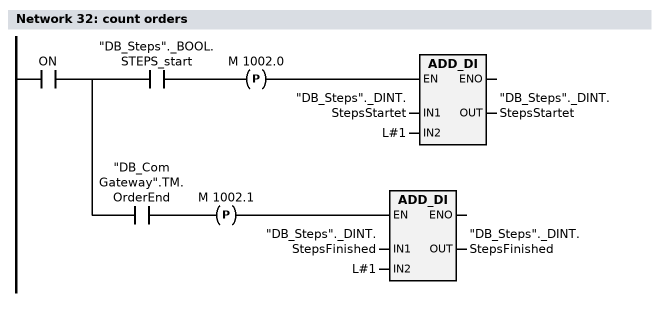
[picture p261: STEPS_OrderData networks 32-32]
NETWORK
TITLE = count orders
      A     "ON";
      =     L 35.0;
      A     L 35.0;
      A(;
      A     "DB_Steps"._BOOL.STEPS_start;
      BLD   100;
      FP    M 1002.0;
      );
      JNB   _01d;
      L     "DB_Steps"._DINT.StepsStartet;
      L     L#1;
      +D;
      T     "DB_Steps"._DINT.StepsStartet;
_01d: NOP   0;
      A     L 35.0;
      A(;
      A     "DB_ComGateway".TM.OrderEnd;
      BLD   100;
      FP    M 1002.1;
      );
      JNB   _01e;
      L     "DB_Steps"._DINT.StepsFinished;
      L     L#1;
      +D;
      T     "DB_Steps"._DINT.StepsFinished;
_01e: NOP   0;
END_FUNCTION

FUNCTION "STEPS_BASEPOS" : VOID	// FC 112
TITLE = Steps BasePos
VERSION : 0.1
BEGIN
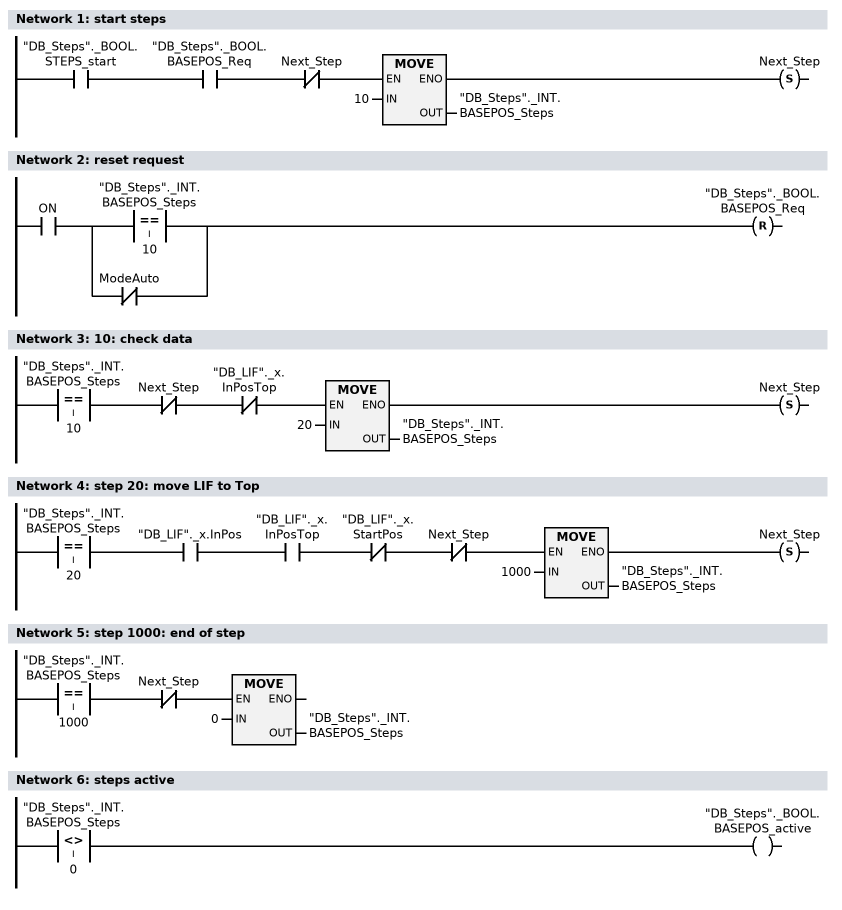
NETWORK
TITLE = start steps
      A     "DB_Steps"._BOOL.STEPS_start;
      A     "DB_Steps"._BOOL.BASEPOS_Req;
      AN    "Next_Step";
      JNB   _001;
      L     10;
      T     "DB_Steps"._INT.BASEPOS_Steps;
      SET;
      SAVE;
      CLR;
_001: A     BR;
      S     "Next_Step";
NETWORK
TITLE = reset request
      A     "ON";
      A(;
      O(;
      L     "DB_Steps"._INT.BASEPOS_Steps;
      L     10;
      ==I;
      );
      ON    "ModeAuto";
      );
      R     "DB_Steps"._BOOL.BASEPOS_Req;
NETWORK
TITLE = 10: check data
//20: move LIF to Top
      A(;
      L     "DB_Steps"._INT.BASEPOS_Steps;
      L     10;
      ==I;
      );
      AN    "Next_Step";
      AN    "DB_LIF"._x.InPosTop;
      JNB   _002;
      L     20;
      T     "DB_Steps"._INT.BASEPOS_Steps;
      SET;
      SAVE;
      CLR;
_002: A     BR;
      S     "Next_Step";
NETWORK
TITLE = step 20: move LIF to Top
//1000: end of steps
      A(;
      L     "DB_Steps"._INT.BASEPOS_Steps;
      L     20;
      ==I;
      );
      A     "DB_LIF"._x.InPos;
      A     "DB_LIF"._x.InPosTop;
      AN    "DB_LIF"._x.StartPos;
      AN    "Next_Step";
      JNB   _003;
      L     1000;
      T     "DB_Steps"._INT.BASEPOS_Steps;
      SET;
      SAVE;
      CLR;
_003: A     BR;
      S     "Next_Step";
NETWORK
TITLE = step 1000: end of step
      A(;
      L     "DB_Steps"._INT.BASEPOS_Steps;
      L     1000;
      ==I;
      );
      AN    "Next_Step";
      JNB   _004;
      L     0;
      T     "DB_Steps"._INT.BASEPOS_Steps;
_004: NOP   0;
NETWORK
TITLE = steps active
      L     "DB_Steps"._INT.BASEPOS_Steps;
      L     0;
      <>I;
      =     "DB_Steps"._BOOL.BASEPOS_active;
END_FUNCTION

FUNCTION "STEPS_EMPTY" : VOID	// FC 113
TITLE = Steps Empty
VERSION : 0.1
BEGIN
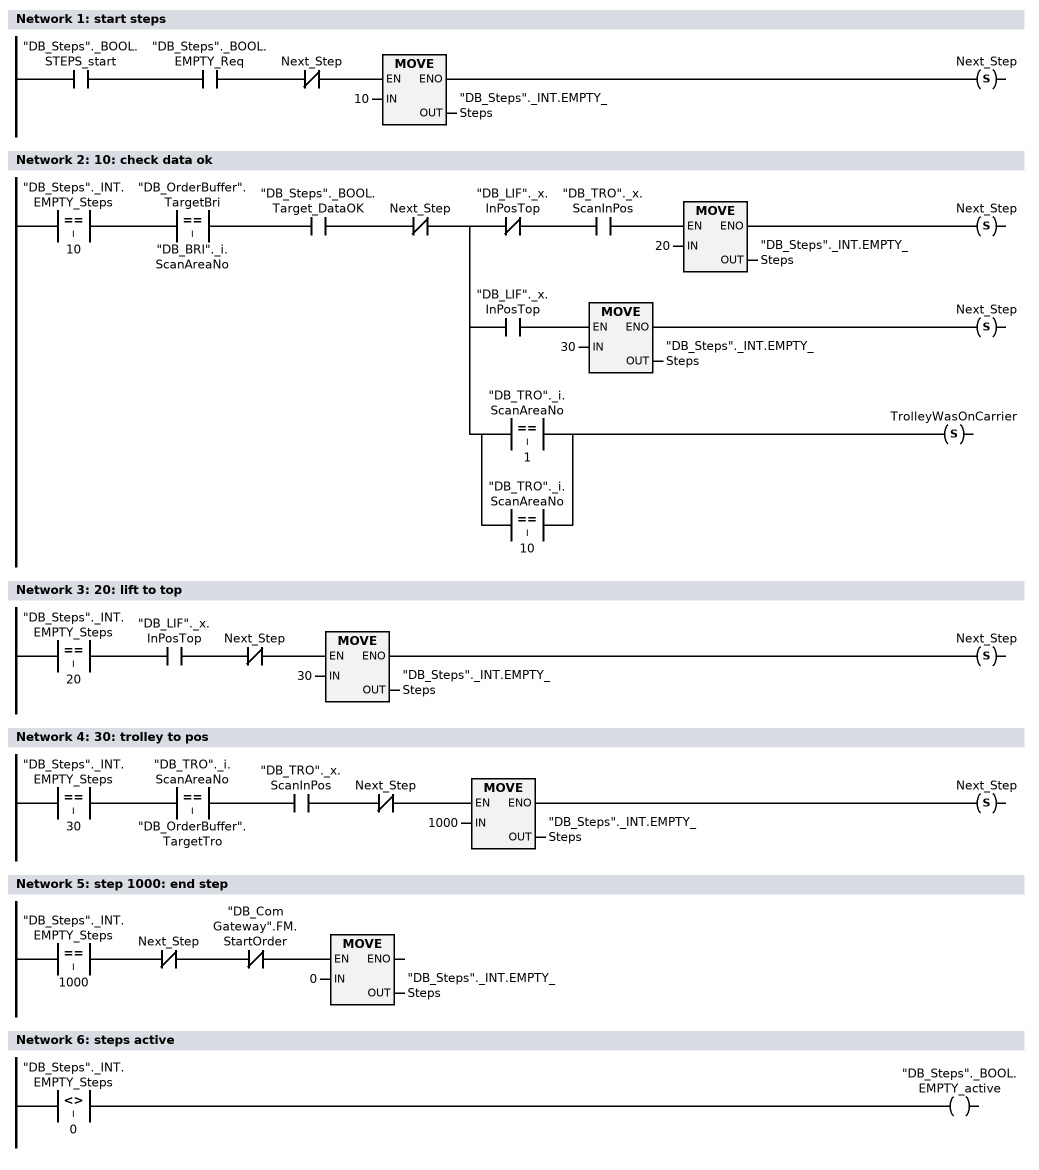
NETWORK
TITLE = start steps
      A     "DB_Steps"._BOOL.STEPS_start;
      A     "DB_Steps"._BOOL.EMPTY_Req;
      AN    "Next_Step";
      JNB   _001;
      L     10;
      T     "DB_Steps"._INT.EMPTY_Steps;
      SET;
      SAVE;
      CLR;
_001: A     BR;
      S     "Next_Step";
NETWORK
TITLE = 10: check data ok
//20: lift to top
//30: BRI to position
      A(;
      L     "DB_Steps"._INT.EMPTY_Steps;
      L     10;
      ==I;
      );
      A(;
      L     "DB_OrderBuffer".TargetBri;
      L     "DB_BRI"._i.ScanAreaNo;
      ==I;
      );
      A     "DB_Steps"._BOOL.Target_DataOK;
      AN    "Next_Step";
      =     L 0.0;
      A     L 0.0;
      AN    "DB_LIF"._x.InPosTop;
      A     "DB_TRO"._x.ScanInPos;
      JNB   _002;
      L     20;
      T     "DB_Steps"._INT.EMPTY_Steps;
      SET;
      SAVE;
      CLR;
_002: A     BR;
      S     "Next_Step";
      A     L 0.0;
      A     "DB_LIF"._x.InPosTop;
      JNB   _003;
      L     30;
      T     "DB_Steps"._INT.EMPTY_Steps;
      SET;
      SAVE;
      CLR;
_003: A     BR;
      S     "Next_Step";
      A     L 0.0;
      A(;
      O(;
      L     "DB_TRO"._i.ScanAreaNo;
      L     1;
      ==I;
      );
      O(;
      L     "DB_TRO"._i.ScanAreaNo;
      L     10;
      ==I;
      );
      );
      S     "TrolleyWasOnCarrier";
NETWORK
TITLE = 20: lift to top
//30: TRO to position
      A(;
      L     "DB_Steps"._INT.EMPTY_Steps;
      L     20;
      ==I;
      );
      A     "DB_LIF"._x.InPosTop;
      AN    "Next_Step";
      JNB   _004;
      L     30;
      T     "DB_Steps"._INT.EMPTY_Steps;
      SET;
      SAVE;
      CLR;
_004: A     BR;
      S     "Next_Step";
NETWORK
TITLE = 30: trolley to pos
      A(;
      L     "DB_Steps"._INT.EMPTY_Steps;
      L     30;
      ==I;
      );
      A(;
      L     "DB_TRO"._i.ScanAreaNo;
      L     "DB_OrderBuffer".TargetTro;
      ==I;
      );
      A     "DB_TRO"._x.ScanInPos;
      AN    "Next_Step";
      JNB   _005;
      L     1000;
      T     "DB_Steps"._INT.EMPTY_Steps;
      SET;
      SAVE;
      CLR;
_005: A     BR;
      S     "Next_Step";
NETWORK
TITLE = step 1000: end step
      A(;
      L     "DB_Steps"._INT.EMPTY_Steps;
      L     1000;
      ==I;
      );
      AN    "Next_Step";
      AN    "DB_ComGateway".FM.StartOrder;
      JNB   _006;
      L     0;
      T     "DB_Steps"._INT.EMPTY_Steps;
_006: NOP   0;
NETWORK
TITLE = steps active
      L     "DB_Steps"._INT.EMPTY_Steps;
      L     0;
      <>I;
      =     "DB_Steps"._BOOL.EMPTY_active;
END_FUNCTION

FUNCTION "STEPS_GET" : VOID	// FC 114
TITLE = Steps GET
VERSION : 0.1
VAR_TEMP
  US_Sensor_OK : BOOL ;
  GetFromLS : BOOL ;
  temp : INT ;
END_VAR
BEGIN
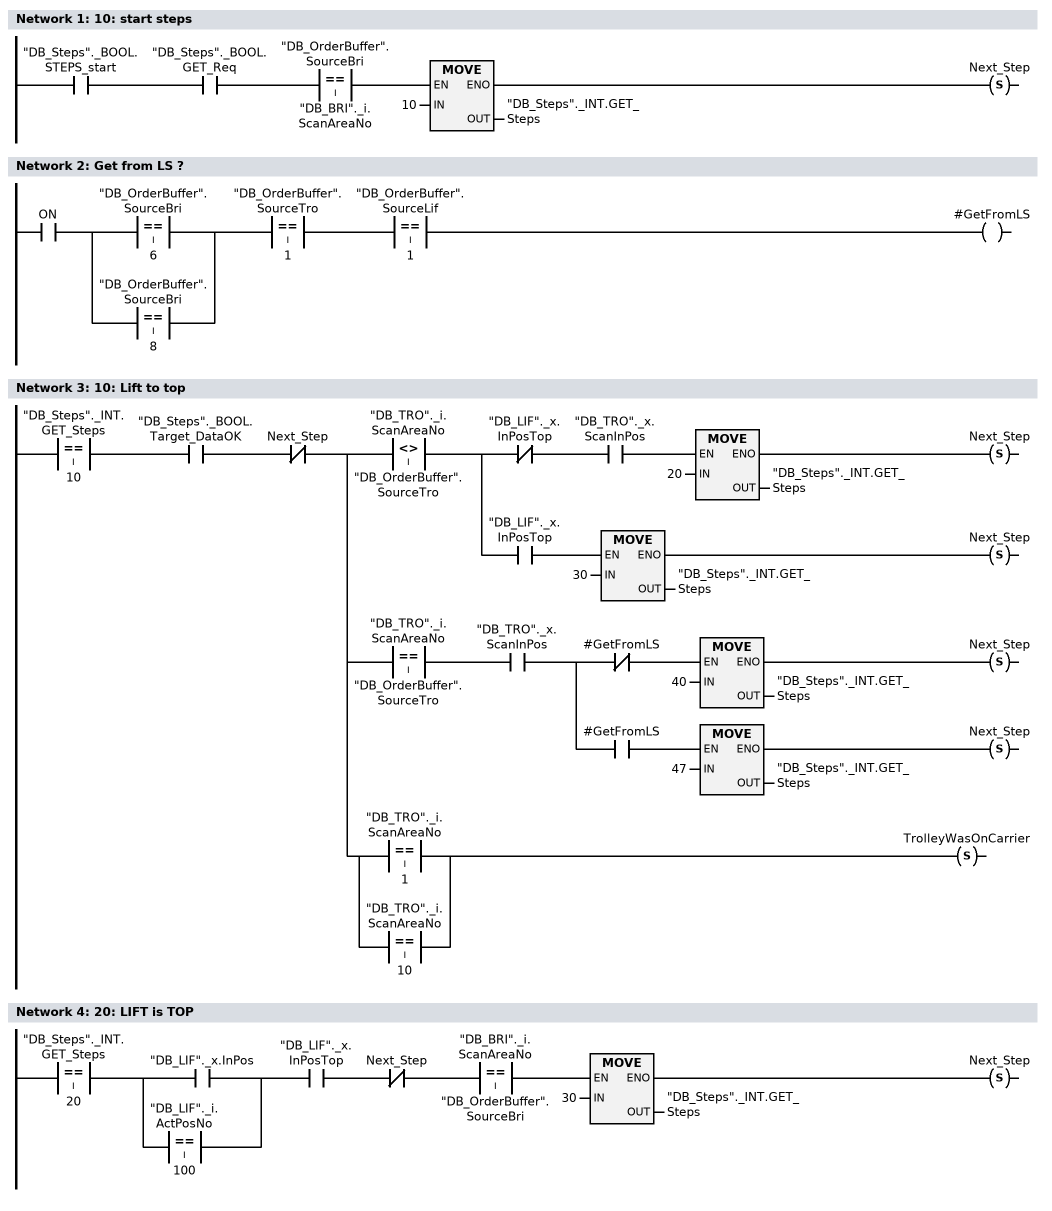
NETWORK
TITLE = 10: start steps
      A     "DB_Steps"._BOOL.STEPS_start;
      A     "DB_Steps"._BOOL.GET_Req;
      A(;
      L     "DB_OrderBuffer".SourceBri;
      L     "DB_BRI"._i.ScanAreaNo;
      ==I;
      );
      JNB   _001;
      L     10;
      T     "DB_Steps"._INT.GET_Steps;
      SET;
      SAVE;
      CLR;
_001: A     BR;
      S     "Next_Step";
NETWORK
TITLE = Get from LS ?
      A     "ON";
      A(;
      O(;
      L     "DB_OrderBuffer".SourceBri;
      L     6;
      ==I;
      );
      O(;
      L     "DB_OrderBuffer".SourceBri;
      L     8;
      ==I;
      );
      );
      A(;
      L     "DB_OrderBuffer".SourceTro;
      L     1;
      ==I;
      );
      A(;
      L     "DB_OrderBuffer".SourceLif;
      L     1;
      ==I;
      );
      =     #GetFromLS;
NETWORK
TITLE = 10: Lift to top
//20: LIF to TOP
//30: BRI to Position
      A(;
      L     "DB_Steps"._INT.GET_Steps;
      L     10;
      ==I;
      );
      A     "DB_Steps"._BOOL.Target_DataOK;
      AN    "Next_Step";
      =     L 4.0;
      A     L 4.0;
      A(;
      L     "DB_TRO"._i.ScanAreaNo;
      L     "DB_OrderBuffer".SourceTro;
      <>I;
      );
      =     L 4.1;
      A     L 4.1;
      AN    "DB_LIF"._x.InPosTop;
      A     "DB_TRO"._x.ScanInPos;
      JNB   _002;
      L     20;
      T     "DB_Steps"._INT.GET_Steps;
      SET;
      SAVE;
      CLR;
_002: A     BR;
      S     "Next_Step";
      A     L 4.1;
      A     "DB_LIF"._x.InPosTop;
      JNB   _003;
      L     30;
      T     "DB_Steps"._INT.GET_Steps;
      SET;
      SAVE;
      CLR;
_003: A     BR;
      S     "Next_Step";
      A     L 4.0;
      A(;
      L     "DB_TRO"._i.ScanAreaNo;
      L     "DB_OrderBuffer".SourceTro;
      ==I;
      );
      A     "DB_TRO"._x.ScanInPos;
      =     L 4.1;
      A     L 4.1;
      AN    #GetFromLS;
      JNB   _004;
      L     40;
      T     "DB_Steps"._INT.GET_Steps;
      SET;
      SAVE;
      CLR;
_004: A     BR;
      S     "Next_Step";
      A     L 4.1;
      A     #GetFromLS;
      JNB   _005;
      L     47;
      T     "DB_Steps"._INT.GET_Steps;
      SET;
      SAVE;
      CLR;
_005: A     BR;
      S     "Next_Step";
      A     L 4.0;
      A(;
      O(;
      L     "DB_TRO"._i.ScanAreaNo;
      L     1;
      ==I;
      );
      O(;
      L     "DB_TRO"._i.ScanAreaNo;
      L     10;
      ==I;
      );
      );
      S     "TrolleyWasOnCarrier";
NETWORK
TITLE = 20: LIFT is TOP
//30: BRI to Position / Start Width S30/S40
      A(;
      L     "DB_Steps"._INT.GET_Steps;
      L     20;
      ==I;
      );
      A(;
      O     "DB_LIF"._x.InPos;
      O(;
      L     "DB_LIF"._i.ActPosNo;
      L     100;
      ==I;
      );
      );
      A     "DB_LIF"._x.InPosTop;
      AN    "Next_Step";
      A(;
      L     "DB_BRI"._i.ScanAreaNo;
      L     "DB_OrderBuffer".SourceBri;
      ==I;
      );
      JNB   _006;
      L     30;
      T     "DB_Steps"._INT.GET_Steps;
      SET;
      SAVE;
      CLR;
_006: A     BR;
      S     "Next_Step";
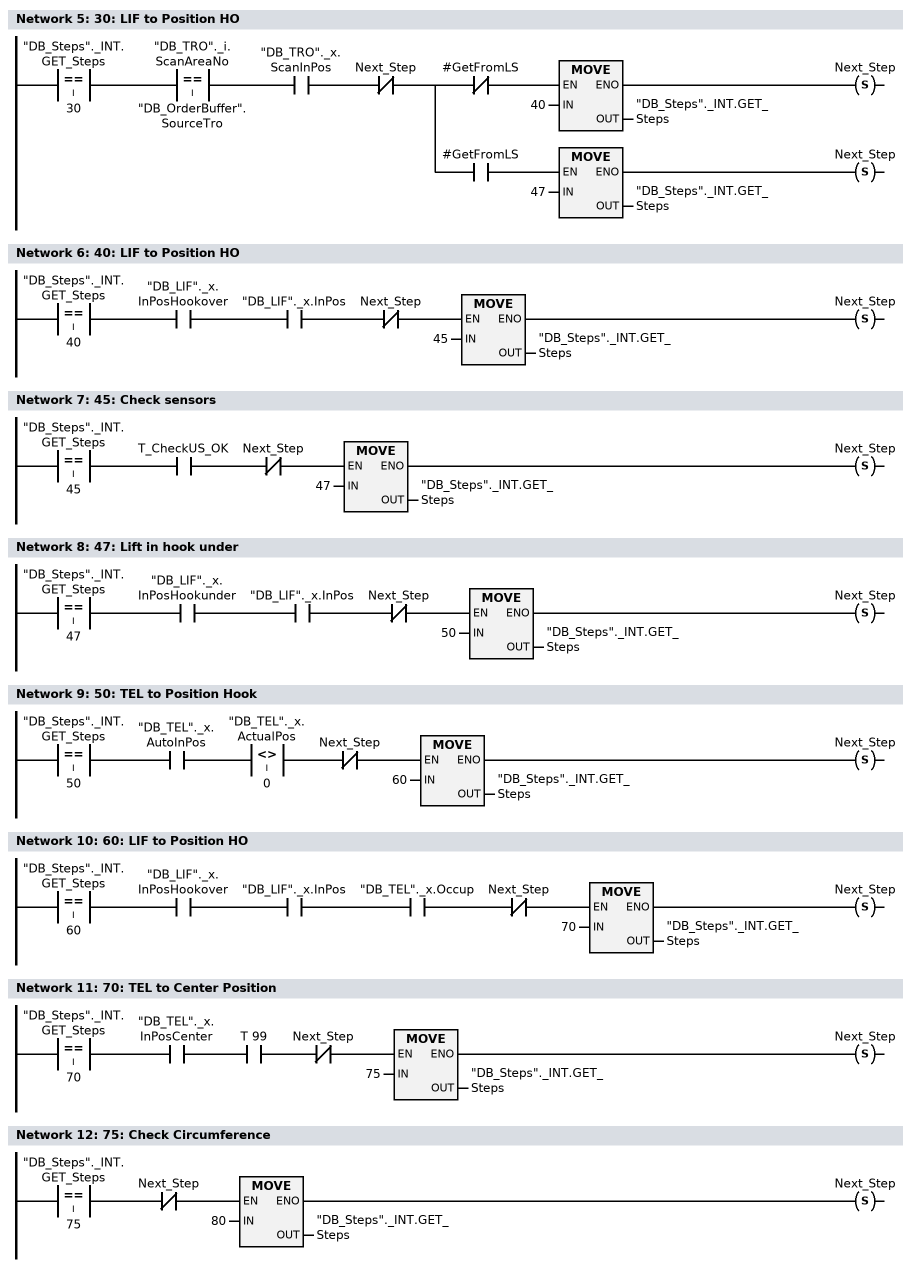
NETWORK
TITLE = 30: LIF to Position HO
      A(;
      L     "DB_Steps"._INT.GET_Steps;
      L     30;
      ==I;
      );
      A(;
      L     "DB_TRO"._i.ScanAreaNo;
      L     "DB_OrderBuffer".SourceTro;
      ==I;
      );
      A     "DB_TRO"._x.ScanInPos;
      AN    "Next_Step";
      =     L 4.0;
      A     L 4.0;
      AN    #GetFromLS;
      JNB   _007;
      L     40;
      T     "DB_Steps"._INT.GET_Steps;
      SET;
      SAVE;
      CLR;
_007: A     BR;
      S     "Next_Step";
      A     L 4.0;
      A     #GetFromLS;
      JNB   _008;
      L     47;
      T     "DB_Steps"._INT.GET_Steps;
      SET;
      SAVE;
      CLR;
_008: A     BR;
      S     "Next_Step";
NETWORK
TITLE = 40: LIF to Position HO
//50: TEL to Position Hook
//45: check occupation sensors hook over
      A(;
      L     "DB_Steps"._INT.GET_Steps;
      L     40;
      ==I;
      );
      A     "DB_LIF"._x.InPosHookover;
      A     "DB_LIF"._x.InPos;
      AN    "Next_Step";
      JNB   _009;
      L     45;
      T     "DB_Steps"._INT.GET_Steps;
      SET;
      SAVE;
      CLR;
_009: A     BR;
      S     "Next_Step";
NETWORK
TITLE = 45: Check sensors
//47: LIF to Position HU
//
//Typ 101 Lager
//Typ 201 Ladestation
//Zyp 299 Buffer
//
//The sensors are not checked on the loading staion
      A(;
      L     "DB_Steps"._INT.GET_Steps;
      L     45;
      ==I;
      );
      A     "T_CheckUS_OK";
      AN    "Next_Step";
      JNB   _00a;
      L     47;
      T     "DB_Steps"._INT.GET_Steps;
      SET;
      SAVE;
      CLR;
_00a: A     BR;
      S     "Next_Step";
NETWORK
TITLE = 47: Lift in hook under
//50: TEL to Position Hook
      A(;
      L     "DB_Steps"._INT.GET_Steps;
      L     47;
      ==I;
      );
      A     "DB_LIF"._x.InPosHookunder;
      A     "DB_LIF"._x.InPos;
      AN    "Next_Step";
      JNB   _00b;
      L     50;
      T     "DB_Steps"._INT.GET_Steps;
      SET;
      SAVE;
      CLR;
_00b: A     BR;
      S     "Next_Step";
NETWORK
TITLE = 50: TEL to Position Hook
//60: LIF to Position HO
      A(;
      L     "DB_Steps"._INT.GET_Steps;
      L     50;
      ==I;
      );
      A     "DB_TEL"._x.AutoInPos;
      A(;
      L     "DB_TEL"._x.ActualPos;
      L     0;
      <>I;
      );
      AN    "Next_Step";
      JNB   _00c;
      L     60;
      T     "DB_Steps"._INT.GET_Steps;
      SET;
      SAVE;
      CLR;
_00c: A     BR;
      S     "Next_Step";
NETWORK
TITLE = 60: LIF to Position HO
//70: TEL to Center Position
      A(;
      L     "DB_Steps"._INT.GET_Steps;
      L     60;
      ==I;
      );
      A     "DB_LIF"._x.InPosHookover;
      A     "DB_LIF"._x.InPos;
      A     "DB_TEL"._x.Occup;
      AN    "Next_Step";
      JNB   _00d;
      L     70;
      T     "DB_Steps"._INT.GET_Steps;
      SET;
      SAVE;
      CLR;
_00d: A     BR;
      S     "Next_Step";
NETWORK
TITLE = 70: TEL to Center Position
//75: Check Circumference
      A(;
      L     "DB_Steps"._INT.GET_Steps;
      L     70;
      ==I;
      );
      A     "DB_TEL"._x.InPosCenter;
      A     T 99;
      AN    "Next_Step";
      JNB   _00e;
      L     75;
      T     "DB_Steps"._INT.GET_Steps;
      SET;
      SAVE;
      CLR;
_00e: A     BR;
      S     "Next_Step";
NETWORK
TITLE = 75: Check Circumference
//510: check hook occupation sensors
// 80: check Lift position safety area loadingstation
      A(;
      L     "DB_Steps"._INT.GET_Steps;
      L     75;
      ==I;
      );
      AN    "Next_Step";
      JNB   _00f;
      L     80;
      T     "DB_Steps"._INT.GET_Steps;
      SET;
      SAVE;
      CLR;
_00f: A     BR;
      S     "Next_Step";
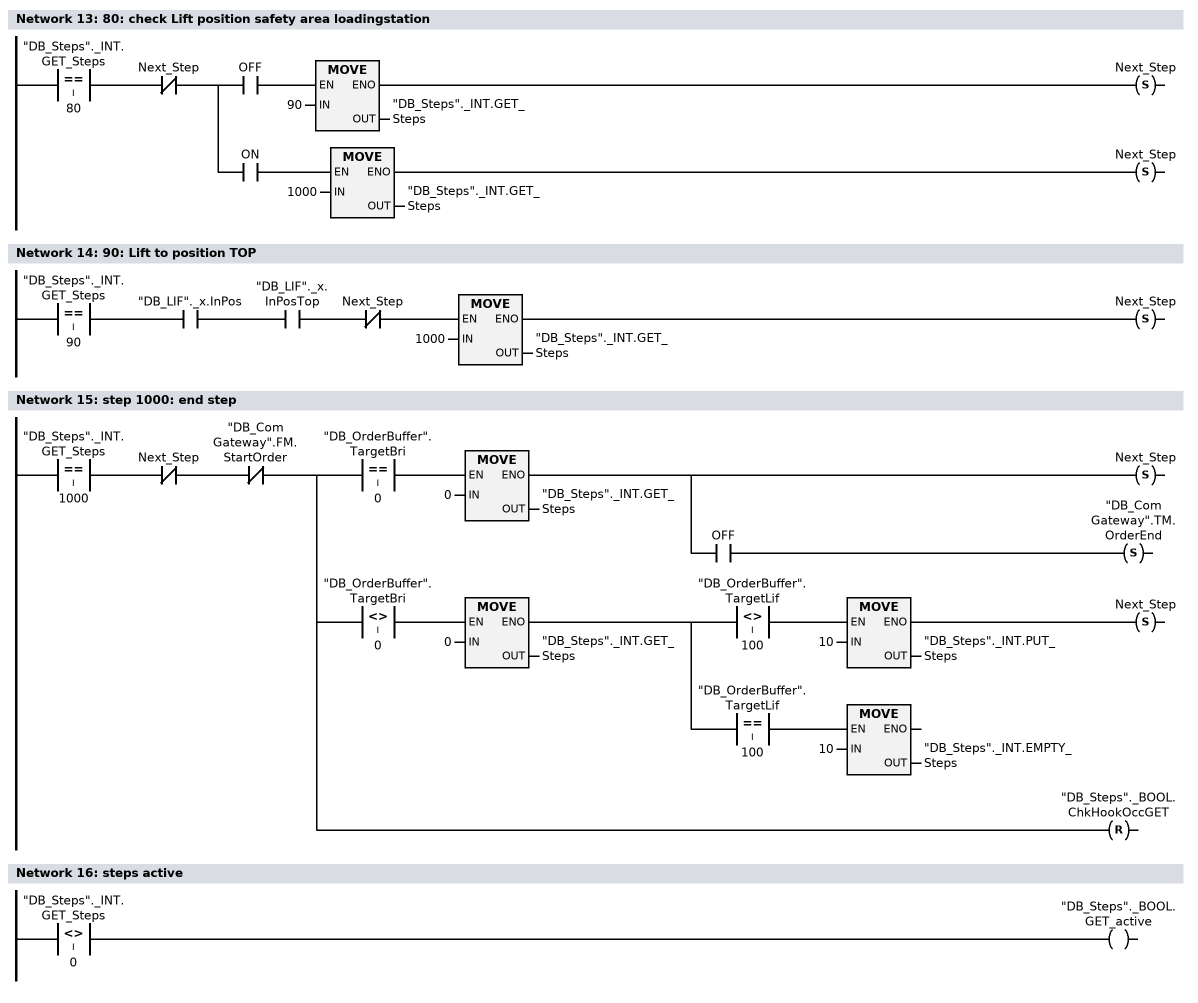
NETWORK
TITLE = 80: check Lift position safety area loadingstation
//85: Get Circumference Value
      A(;
      L     "DB_Steps"._INT.GET_Steps;
      L     80;
      ==I;
      );
      AN    "Next_Step";
      =     L 4.0;
      A     L 4.0;
      A     "OFF";
      JNB   _010;
      L     90;
      T     "DB_Steps"._INT.GET_Steps;
      SET;
      SAVE;
      CLR;
_010: A     BR;
      S     "Next_Step";
      A     L 4.0;
      A     "ON";
      JNB   _011;
      L     1000;
      T     "DB_Steps"._INT.GET_Steps;
      SET;
      SAVE;
      CLR;
_011: A     BR;
      S     "Next_Step";
NETWORK
TITLE = 90: Lift to position TOP
      A(;
      L     "DB_Steps"._INT.GET_Steps;
      L     90;
      ==I;
      );
      A     "DB_LIF"._x.InPos;
      A     "DB_LIF"._x.InPosTop;
      AN    "Next_Step";
      JNB   _012;
      L     1000;
      T     "DB_Steps"._INT.GET_Steps;
      SET;
      SAVE;
      CLR;
_012: A     BR;
      S     "Next_Step";
NETWORK
TITLE = step 1000: end step
      A(;
      L     "DB_Steps"._INT.GET_Steps;
      L     1000;
      ==I;
      );
      AN    "Next_Step";
      AN    "DB_ComGateway".FM.StartOrder;
      =     L 4.0;
      A     L 4.0;
      A(;
      L     "DB_OrderBuffer".TargetBri;
      L     0;
      ==I;
      );
      JNB   _013;
      L     0;
      T     "DB_Steps"._INT.GET_Steps;
      SET;
      SAVE;
      CLR;
_013: A     BR;
      =     L 4.1;
      A     L 4.1;
      BLD   102;
      S     "Next_Step";
      A     L 4.1;
      A     "OFF";
      S     "DB_ComGateway".TM.OrderEnd;
      A     L 4.0;
      A(;
      L     "DB_OrderBuffer".TargetBri;
      L     0;
      <>I;
      );
      JNB   _014;
      L     0;
      T     "DB_Steps"._INT.GET_Steps;
      SET;
      SAVE;
      CLR;
_014: A     BR;
      =     L 4.1;
      A     L 4.1;
      A(;
      L     "DB_OrderBuffer".TargetLif;
      L     100;
      <>I;
      );
      JNB   _015;
      L     10;
      T     "DB_Steps"._INT.PUT_Steps;
      SET;
      SAVE;
      CLR;
_015: A     BR;
      S     "Next_Step";
      A     L 4.1;
      A(;
      L     "DB_OrderBuffer".TargetLif;
      L     100;
      ==I;
      );
      JNB   _016;
      L     10;
      T     "DB_Steps"._INT.EMPTY_Steps;
_016: NOP   0;
      A     L 4.0;
      BLD   102;
      R     "DB_Steps"._BOOL.ChkHookOccGET;
NETWORK
TITLE = steps active
      L     "DB_Steps"._INT.GET_Steps;
      L     0;
      <>I;
      =     "DB_Steps"._BOOL.GET_active;
END_FUNCTION

FUNCTION "STEPS_PUT" : VOID	// FC 115
TITLE = Steps PUT
VERSION : 0.1
VAR_TEMP
  US_Sensor_OK : BOOL ;
  PutToLS : BOOL ;
  temp : INT ;
END_VAR
BEGIN
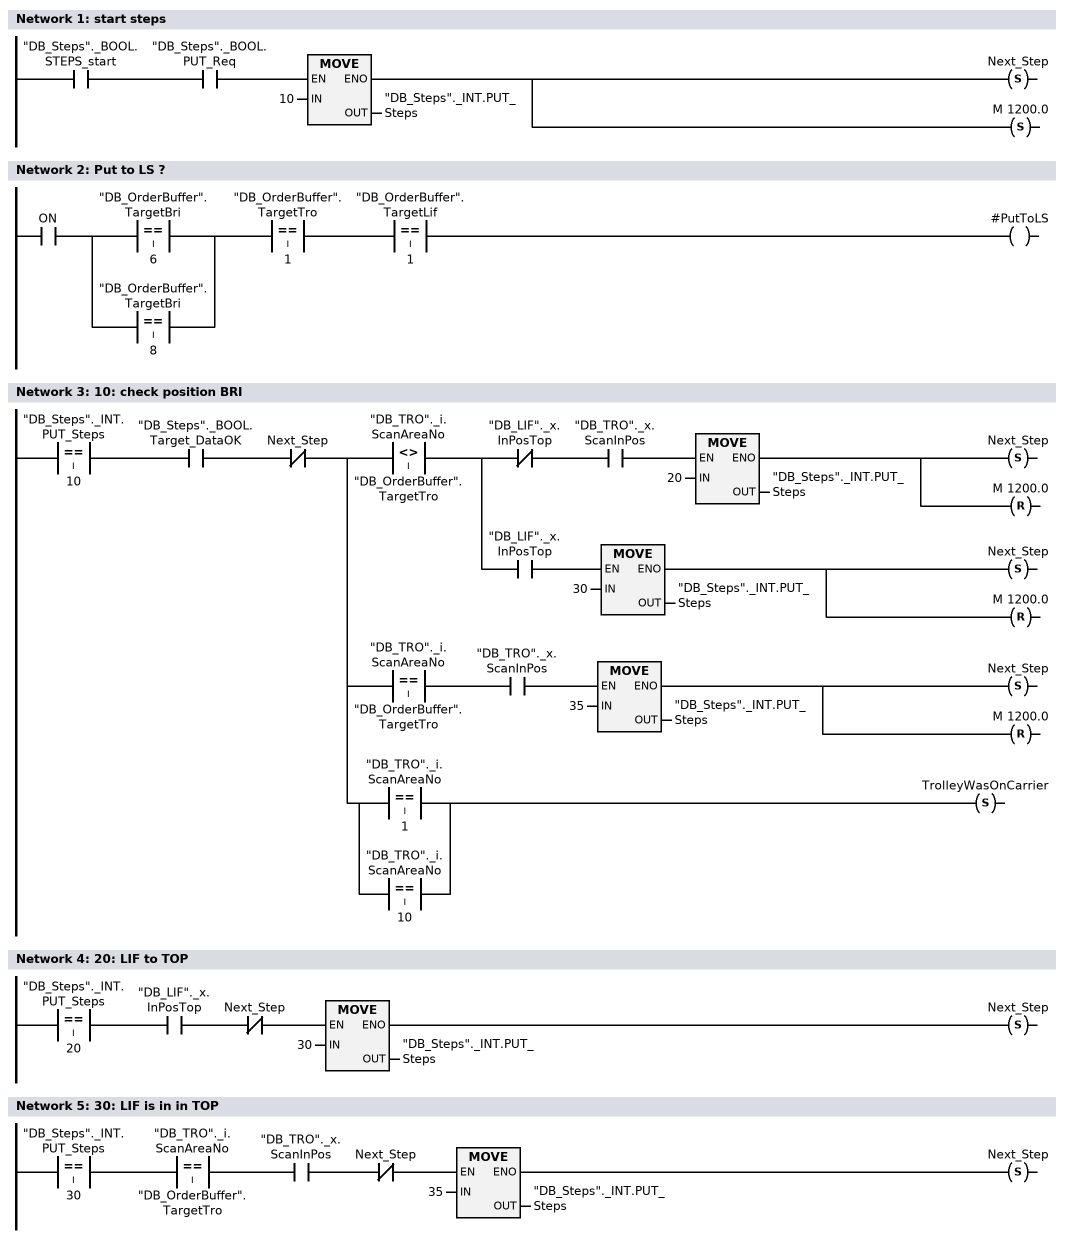
NETWORK
TITLE = start steps
      A     "DB_Steps"._BOOL.STEPS_start;
      A     "DB_Steps"._BOOL.PUT_Req;
      JNB   _001;
      L     10;
      T     "DB_Steps"._INT.PUT_Steps;
      SET;
      SAVE;
      CLR;
_001: A     BR;
      S     "Next_Step";
      S     M 1200.0;
NETWORK
TITLE = Put to LS ?
      A     "ON";
      A(;
      O(;
      L     "DB_OrderBuffer".TargetBri;
      L     6;
      ==I;
      );
      O(;
      L     "DB_OrderBuffer".TargetBri;
      L     8;
      ==I;
      );
      );
      A(;
      L     "DB_OrderBuffer".TargetTro;
      L     1;
      ==I;
      );
      A(;
      L     "DB_OrderBuffer".TargetLif;
      L     1;
      ==I;
      );
      =     #PutToLS;
NETWORK
TITLE = 10: check position BRI
//20: LIF to TOP
//30: BRI to Position
      A(;
      L     "DB_Steps"._INT.PUT_Steps;
      L     10;
      ==I;
      );
      A     "DB_Steps"._BOOL.Target_DataOK;
      AN    "Next_Step";
      =     L 4.0;
      A     L 4.0;
      A(;
      L     "DB_TRO"._i.ScanAreaNo;
      L     "DB_OrderBuffer".TargetTro;
      <>I;
      );
      =     L 4.1;
      A     L 4.1;
      AN    "DB_LIF"._x.InPosTop;
      A     "DB_TRO"._x.ScanInPos;
      JNB   _002;
      L     20;
      T     "DB_Steps"._INT.PUT_Steps;
      SET;
      SAVE;
      CLR;
_002: A     BR;
      S     "Next_Step";
      R     M 1200.0;
      A     L 4.1;
      A     "DB_LIF"._x.InPosTop;
      JNB   _003;
      L     30;
      T     "DB_Steps"._INT.PUT_Steps;
      SET;
      SAVE;
      CLR;
_003: A     BR;
      S     "Next_Step";
      R     M 1200.0;
      A     L 4.0;
      A(;
      L     "DB_TRO"._i.ScanAreaNo;
      L     "DB_OrderBuffer".TargetTro;
      ==I;
      );
      A     "DB_TRO"._x.ScanInPos;
      JNB   _004;
      L     35;
      T     "DB_Steps"._INT.PUT_Steps;
      SET;
      SAVE;
      CLR;
_004: A     BR;
      S     "Next_Step";
      R     M 1200.0;
      A     L 4.0;
      A(;
      O(;
      L     "DB_TRO"._i.ScanAreaNo;
      L     1;
      ==I;
      );
      O(;
      L     "DB_TRO"._i.ScanAreaNo;
      L     10;
      ==I;
      );
      );
      S     "TrolleyWasOnCarrier";
NETWORK
TITLE = 20: LIF to TOP
//30: BRI to Position
      A(;
      L     "DB_Steps"._INT.PUT_Steps;
      L     20;
      ==I;
      );
      A     "DB_LIF"._x.InPosTop;
      AN    "Next_Step";
      JNB   _005;
      L     30;
      T     "DB_Steps"._INT.PUT_Steps;
      SET;
      SAVE;
      CLR;
_005: A     BR;
      S     "Next_Step";
NETWORK
TITLE = 30: LIF is in in TOP
//35: LIF to Position HO
      A(;
      L     "DB_Steps"._INT.PUT_Steps;
      L     30;
      ==I;
      );
      A(;
      L     "DB_TRO"._i.ScanAreaNo;
      L     "DB_OrderBuffer".TargetTro;
      ==I;
      );
      A     "DB_TRO"._x.ScanInPos;
      AN    "Next_Step";
      JNB   _006;
      L     35;
      T     "DB_Steps"._INT.PUT_Steps;
      SET;
      SAVE;
      CLR;
_006: A     BR;
      S     "Next_Step";
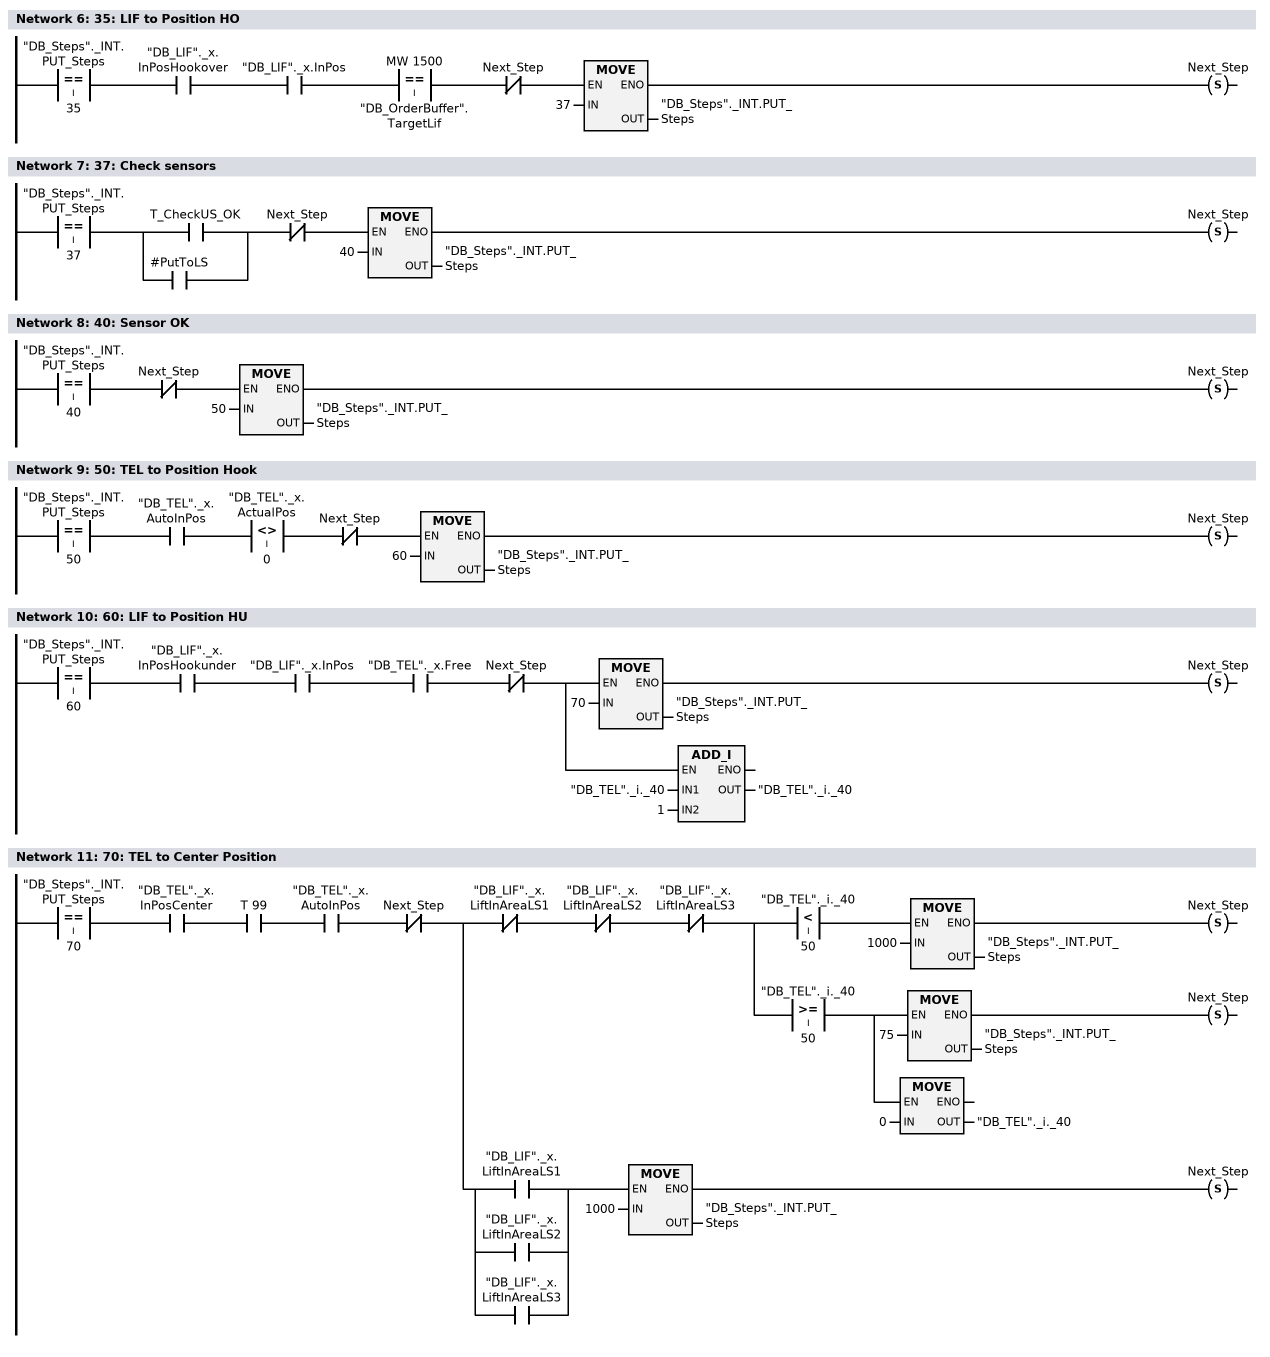
NETWORK
TITLE = 35: LIF to Position HO
//50: TEL to Position Hook
      A(;
      L     "DB_Steps"._INT.PUT_Steps;
      L     35;
      ==I;
      );
      A     "DB_LIF"._x.InPosHookover;
      A     "DB_LIF"._x.InPos;
      A(;
      L     MW 1500;
      L     "DB_OrderBuffer".TargetLif;
      ==I;
      );
      AN    "Next_Step";
      JNB   _007;
      L     37;
      T     "DB_Steps"._INT.PUT_Steps;
      SET;
      SAVE;
      CLR;
_007: A     BR;
      S     "Next_Step";
NETWORK
TITLE = 37: Check sensors
//50: TEL to Position Hook
      A(;
      L     "DB_Steps"._INT.PUT_Steps;
      L     37;
      ==I;
      );
      A(;
      O     "T_CheckUS_OK";
      O     #PutToLS;
      );
      AN    "Next_Step";
      JNB   _008;
      L     40;
      T     "DB_Steps"._INT.PUT_Steps;
      SET;
      SAVE;
      CLR;
_008: A     BR;
      S     "Next_Step";
NETWORK
TITLE = 40: Sensor OK
//50: TEL to Position Hook
      A(;
      L     "DB_Steps"._INT.PUT_Steps;
      L     40;
      ==I;
      );
      AN    "Next_Step";
      JNB   _009;
      L     50;
      T     "DB_Steps"._INT.PUT_Steps;
      SET;
      SAVE;
      CLR;
_009: A     BR;
      S     "Next_Step";
NETWORK
TITLE = 50: TEL to Position Hook
//60: LIF to Position HU
      A(;
      L     "DB_Steps"._INT.PUT_Steps;
      L     50;
      ==I;
      );
      A     "DB_TEL"._x.AutoInPos;
      A(;
      L     "DB_TEL"._x.ActualPos;
      L     0;
      <>I;
      );
      AN    "Next_Step";
      JNB   _00a;
      L     60;
      T     "DB_Steps"._INT.PUT_Steps;
      SET;
      SAVE;
      CLR;
_00a: A     BR;
      S     "Next_Step";
NETWORK
TITLE = 60: LIF to Position HU
//70: TEL to Center Position
      A(;
      L     "DB_Steps"._INT.PUT_Steps;
      L     60;
      ==I;
      );
      A     "DB_LIF"._x.InPosHookunder;
      A     "DB_LIF"._x.InPos;
      A     "DB_TEL"._x.Free;
      AN    "Next_Step";
      =     L 4.0;
      A     L 4.0;
      JNB   _00b;
      L     70;
      T     "DB_Steps"._INT.PUT_Steps;
      SET;
      SAVE;
      CLR;
_00b: A     BR;
      S     "Next_Step";
      A     L 4.0;
      JNB   _00c;
      L     "DB_TEL"._i._40;
      L     1;
      +I;
      T     "DB_TEL"._i._40;
_00c: NOP   0;
NETWORK
TITLE = 70: TEL to Center Position
//75: check occupation sensors hook
      A(;
      L     "DB_Steps"._INT.PUT_Steps;
      L     70;
      ==I;
      );
      A     "DB_TEL"._x.InPosCenter;
      A     T 99;
      A     "DB_TEL"._x.AutoInPos;
      AN    "Next_Step";
      =     L 4.0;
      A     L 4.0;
      AN    "DB_LIF"._x.LiftInAreaLS1;
      AN    "DB_LIF"._x.LiftInAreaLS2;
      AN    "DB_LIF"._x.LiftInAreaLS3;
      =     L 4.1;
      A     L 4.1;
      A(;
      L     "DB_TEL"._i._40;
      L     50;
      <I;
      );
      JNB   _00d;
      L     1000;
      T     "DB_Steps"._INT.PUT_Steps;
      SET;
      SAVE;
      CLR;
_00d: A     BR;
      S     "Next_Step";
      A     L 4.1;
      A(;
      L     "DB_TEL"._i._40;
      L     50;
      >=I;
      );
      =     L 4.2;
      A     L 4.2;
      JNB   _00e;
      L     75;
      T     "DB_Steps"._INT.PUT_Steps;
      SET;
      SAVE;
      CLR;
_00e: A     BR;
      S     "Next_Step";
      A     L 4.2;
      JNB   _00f;
      L     0;
      T     "DB_TEL"._i._40;
_00f: NOP   0;
      A     L 4.0;
      A(;
      O     "DB_LIF"._x.LiftInAreaLS1;
      O     "DB_LIF"._x.LiftInAreaLS2;
      O     "DB_LIF"._x.LiftInAreaLS3;
      );
      JNB   _010;
      L     1000;
      T     "DB_Steps"._INT.PUT_Steps;
      SET;
      SAVE;
      CLR;
_010: A     BR;
      S     "Next_Step";
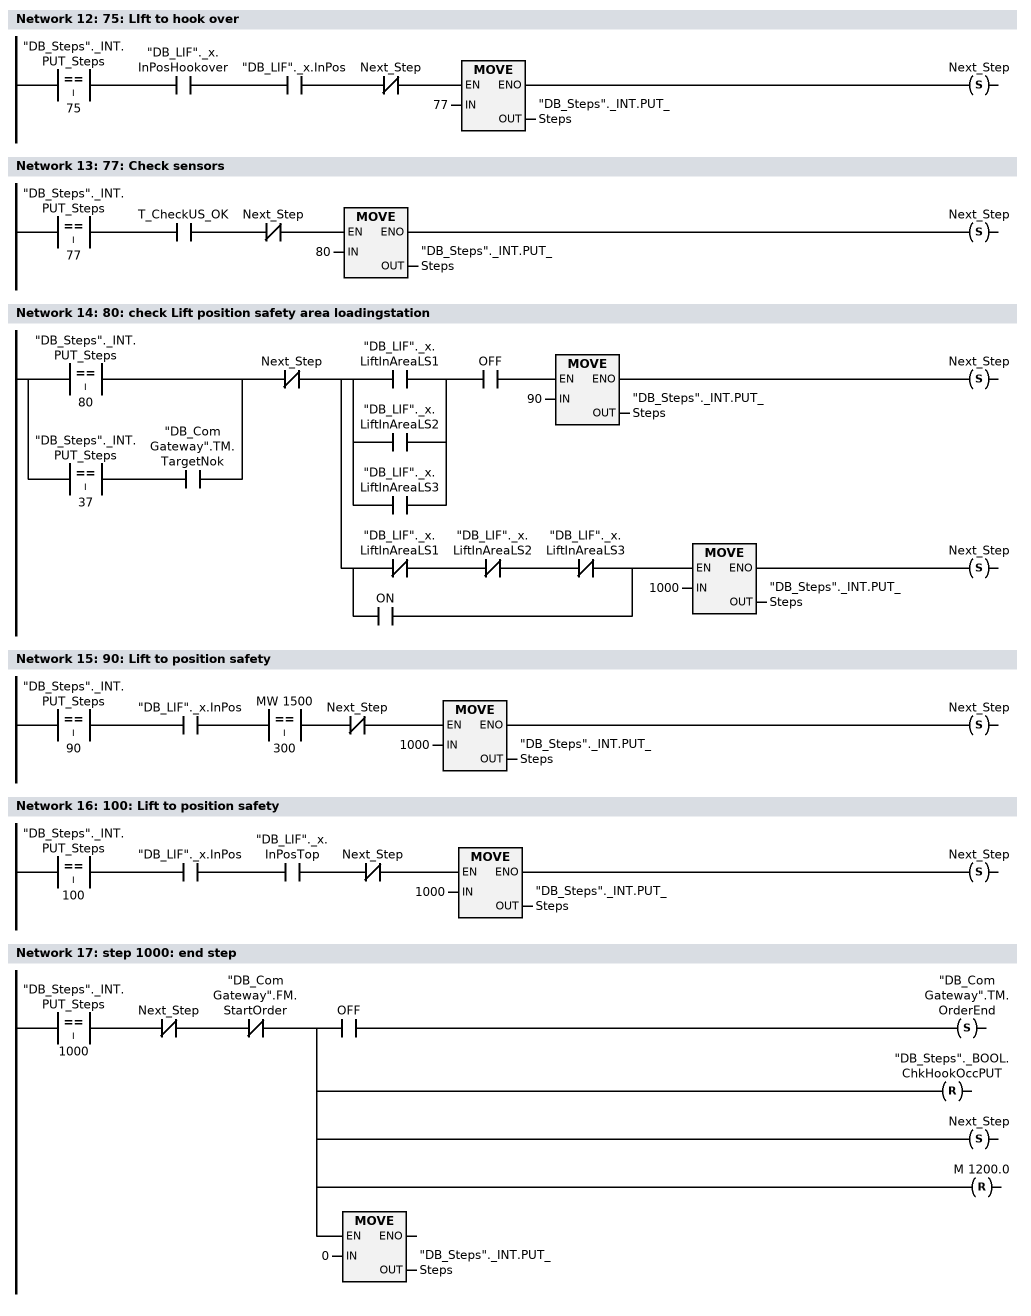
NETWORK
TITLE = 75: LIft to hook over
      A(;
      L     "DB_Steps"._INT.PUT_Steps;
      L     75;
      ==I;
      );
      A     "DB_LIF"._x.InPosHookover;
      A     "DB_LIF"._x.InPos;
      AN    "Next_Step";
      JNB   _011;
      L     77;
      T     "DB_Steps"._INT.PUT_Steps;
      SET;
      SAVE;
      CLR;
_011: A     BR;
      S     "Next_Step";
NETWORK
TITLE = 77: Check sensors
//80: Check Lift position
      A(;
      L     "DB_Steps"._INT.PUT_Steps;
      L     77;
      ==I;
      );
      A     "T_CheckUS_OK";
      AN    "Next_Step";
      JNB   _012;
      L     80;
      T     "DB_Steps"._INT.PUT_Steps;
      SET;
      SAVE;
      CLR;
_012: A     BR;
      S     "Next_Step";
NETWORK
TITLE = 80: check Lift position safety area loadingstation
//90: Lift to position TOP
      A(;
      O(;
      L     "DB_Steps"._INT.PUT_Steps;
      L     80;
      ==I;
      );
      O;
      A(;
      L     "DB_Steps"._INT.PUT_Steps;
      L     37;
      ==I;
      );
      A     "DB_ComGateway".TM.TargetNok;
      );
      AN    "Next_Step";
      =     L 4.0;
      A     L 4.0;
      A(;
      O     "DB_LIF"._x.LiftInAreaLS1;
      O     "DB_LIF"._x.LiftInAreaLS2;
      O     "DB_LIF"._x.LiftInAreaLS3;
      );
      A     "OFF";
      JNB   _013;
      L     90;
      T     "DB_Steps"._INT.PUT_Steps;
      SET;
      SAVE;
      CLR;
_013: A     BR;
      S     "Next_Step";
      A     L 4.0;
      A(;
      AN    "DB_LIF"._x.LiftInAreaLS1;
      AN    "DB_LIF"._x.LiftInAreaLS2;
      AN    "DB_LIF"._x.LiftInAreaLS3;
      O     "ON";
      );
      JNB   _014;
      L     1000;
      T     "DB_Steps"._INT.PUT_Steps;
      SET;
      SAVE;
      CLR;
_014: A     BR;
      S     "Next_Step";
NETWORK
TITLE = 90: Lift to position safety
      A(;
      L     "DB_Steps"._INT.PUT_Steps;
      L     90;
      ==I;
      );
      A     "DB_LIF"._x.InPos;
      A(;
      L     MW 1500;
      L     300;
      ==I;
      );
      AN    "Next_Step";
      JNB   _015;
      L     1000;
      T     "DB_Steps"._INT.PUT_Steps;
      SET;
      SAVE;
      CLR;
_015: A     BR;
      S     "Next_Step";
NETWORK
TITLE = 100: Lift to position safety
      A(;
      L     "DB_Steps"._INT.PUT_Steps;
      L     100;
      ==I;
      );
      A     "DB_LIF"._x.InPos;
      A     "DB_LIF"._x.InPosTop;
      AN    "Next_Step";
      JNB   _016;
      L     1000;
      T     "DB_Steps"._INT.PUT_Steps;
      SET;
      SAVE;
      CLR;
_016: A     BR;
      S     "Next_Step";
NETWORK
TITLE = step 1000: end step
      A(;
      L     "DB_Steps"._INT.PUT_Steps;
      L     1000;
      ==I;
      );
      AN    "Next_Step";
      AN    "DB_ComGateway".FM.StartOrder;
      =     L 4.0;
      A     L 4.0;
      A     "OFF";
      S     "DB_ComGateway".TM.OrderEnd;
      A     L 4.0;
      BLD   102;
      R     "DB_Steps"._BOOL.ChkHookOccPUT;
      A     L 4.0;
      BLD   102;
      S     "Next_Step";
      A     L 4.0;
      BLD   102;
      R     M 1200.0;
      A     L 4.0;
      JNB   _017;
      L     0;
      T     "DB_Steps"._INT.PUT_Steps;
_017: NOP   0;
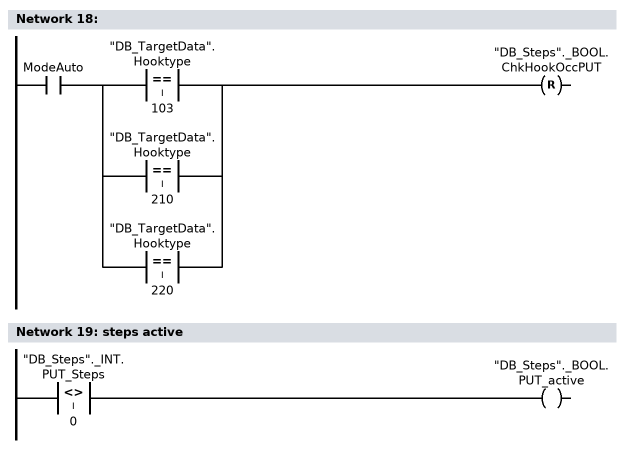
NETWORK
TITLE =
      A     "ModeAuto";
      A(;
      O(;
      L     "DB_TargetData".Hooktype;
      L     103;
      ==I;
      );
      O(;
      L     "DB_TargetData".Hooktype;
      L     210;
      ==I;
      );
      O(;
      L     "DB_TargetData".Hooktype;
      L     220;
      ==I;
      );
      );
      R     "DB_Steps"._BOOL.ChkHookOccPUT;
NETWORK
TITLE = steps active
      L     "DB_Steps"._INT.PUT_Steps;
      L     0;
      <>I;
      =     "DB_Steps"._BOOL.PUT_active;
END_FUNCTION

FUNCTION "Axis_TROLLEY" : VOID	// FC 210
TITLE = Axis TROLLEY
VERSION : 0.1
BEGIN
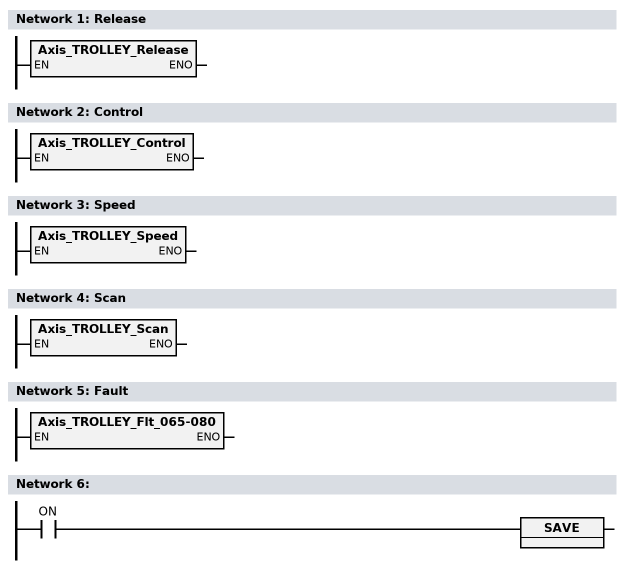
NETWORK
TITLE = Release
      CALL  "Axis_TROLLEY_Release";
      NOP   0;
NETWORK
TITLE = Control
      CALL  "Axis_TROLLEY_Control";
      NOP   0;
NETWORK
TITLE = Speed
      CALL  "Axis_TROLLEY_Speed";
      NOP   0;
NETWORK
TITLE = Scan
      CALL  "Axis_TROLLEY_Scan";
      NOP   0;
NETWORK
TITLE = Fault
      CALL  "Axis_TROLLEY_Flt_065-080";
      NOP   0;
NETWORK
TITLE =
      A     "ON";
      SAVE;
END_FUNCTION

FUNCTION "Axis_TROLLEY_Release" : VOID	// FC 211
TITLE = Axis Trolley Release
//TODO Release if driving to/from carrier (no value)
VERSION : 0.1
BEGIN
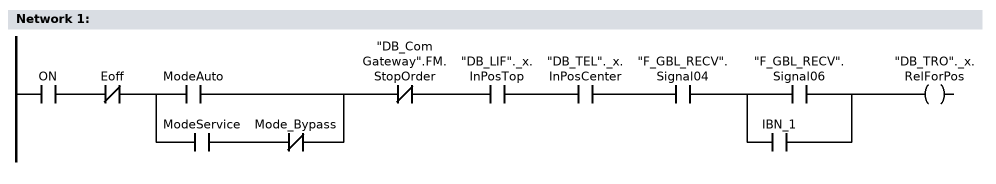
NETWORK
TITLE =
      A     "ON";
      AN    "Eoff";
      A(;
      O     "ModeAuto";
      O;
      A     "ModeService";
      AN    "Mode_Bypass";
      );
      AN    "DB_ComGateway".FM.StopOrder;
      A     "DB_LIF"._x.InPosTop;
      A     "DB_TEL"._x.InPosCenter;
      A     "F_GBL_RECV".Signal04;
      A(;
      O     "F_GBL_RECV".Signal06;
      O     "IBN_1";
      );
      =     "DB_TRO"._x.RelForPos;
END_FUNCTION

FUNCTION "Axis_TROLLEY_Control" : VOID	// FC 212
TITLE = TROLLEY Control
VERSION : 0.1
VAR_TEMP
  PositionMode : BOOL ;
  tmp_TagetPos_Auto : BOOL ;
  tmp_TagetPos_Manual : BOOL ;
  tmp_TargetValueOK : BOOL ;
  mode_ref : BOOL ;
  getValue : BOOL ;
  modeService : BOOL ;
  modeEmergency : BOOL ;
  db_no : INT ;
  prev : DINT ;
  next : DINT ;
  min : DINT ;
  max : DINT ;
  Error : WORD ;
END_VAR
BEGIN
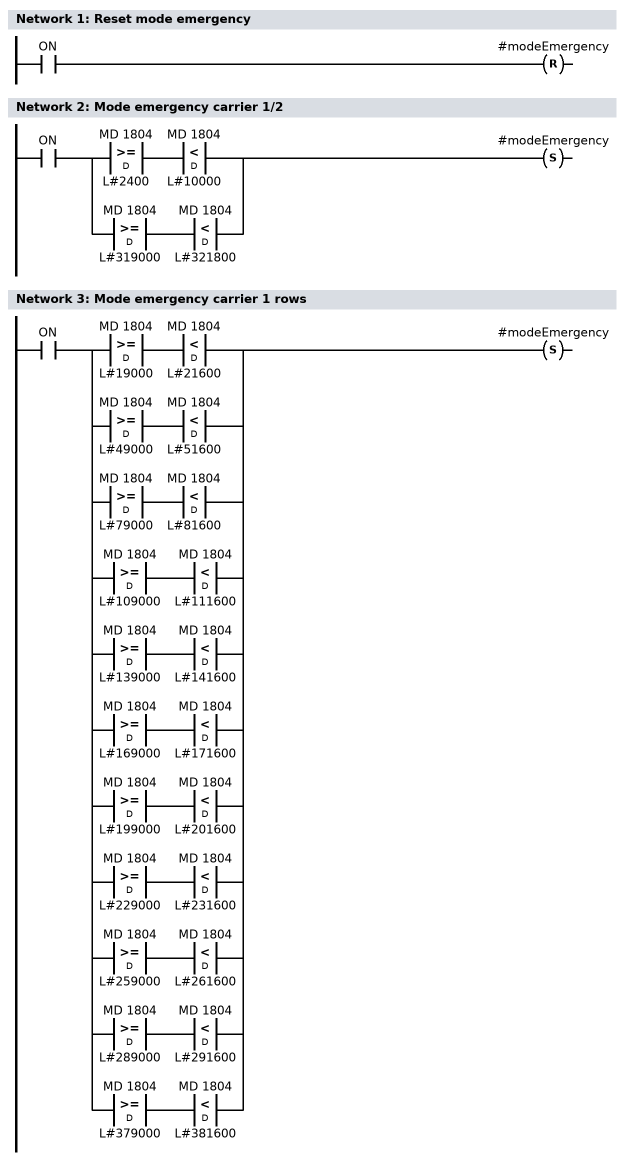
NETWORK
TITLE = Reset mode emergency
      A     "ON";
      R     #modeEmergency;
NETWORK
TITLE = Mode emergency carrier 1/2
      A     "ON";
      A(;
      A(;
      L     MD 1804;
      L     L#2400;
      >=D;
      );
      A(;
      L     MD 1804;
      L     L#10000;
      <D;
      );
      O;
      A(;
      L     MD 1804;
      L     L#319000;
      >=D;
      );
      A(;
      L     MD 1804;
      L     L#321800;
      <D;
      );
      );
      S     #modeEmergency;
NETWORK
TITLE = Mode emergency carrier 1 rows
      A     "ON";
      A(;
      A(;
      L     MD 1804;
      L     L#19000;
      >=D;
      );
      A(;
      L     MD 1804;
      L     L#21600;
      <D;
      );
      O;
      A(;
      L     MD 1804;
      L     L#49000;
      >=D;
      );
      A(;
      L     MD 1804;
      L     L#51600;
      <D;
      );
      O;
      A(;
      L     MD 1804;
      L     L#79000;
      >=D;
      );
      A(;
      L     MD 1804;
      L     L#81600;
      <D;
      );
      O;
      A(;
      L     MD 1804;
      L     L#109000;
      >=D;
      );
      A(;
      L     MD 1804;
      L     L#111600;
      <D;
      );
      O;
      A(;
      L     MD 1804;
      L     L#139000;
      >=D;
      );
      A(;
      L     MD 1804;
      L     L#141600;
      <D;
      );
      O;
      A(;
      L     MD 1804;
      L     L#169000;
      >=D;
      );
      A(;
      L     MD 1804;
      L     L#171600;
      <D;
      );
      O;
      A(;
      L     MD 1804;
      L     L#199000;
      >=D;
      );
      A(;
      L     MD 1804;
      L     L#201600;
      <D;
      );
      O;
      A(;
      L     MD 1804;
      L     L#229000;
      >=D;
      );
      A(;
      L     MD 1804;
      L     L#231600;
      <D;
      );
      O;
      A(;
      L     MD 1804;
      L     L#259000;
      >=D;
      );
      A(;
      L     MD 1804;
      L     L#261600;
      <D;
      );
      O;
      A(;
      L     MD 1804;
      L     L#289000;
      >=D;
      );
      A(;
      L     MD 1804;
      L     L#291600;
      <D;
      );
      O;
      A(;
      L     MD 1804;
      L     L#379000;
      >=D;
      );
      A(;
      L     MD 1804;
      L     L#381600;
      <D;
      );
      );
      S     #modeEmergency;
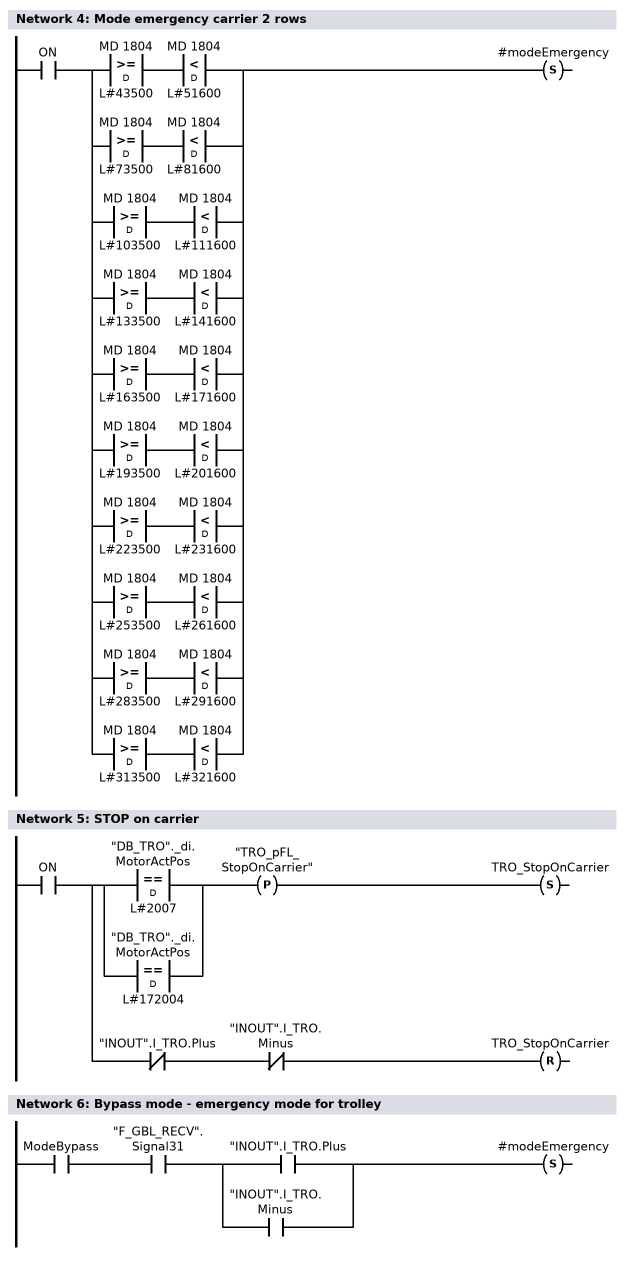
NETWORK
TITLE = Mode emergency carrier 2 rows
      A     "ON";
      A(;
      A(;
      L     MD 1804;
      L     L#43500;
      >=D;
      );
      A(;
      L     MD 1804;
      L     L#51600;
      <D;
      );
      O;
      A(;
      L     MD 1804;
      L     L#73500;
      >=D;
      );
      A(;
      L     MD 1804;
      L     L#81600;
      <D;
      );
      O;
      A(;
      L     MD 1804;
      L     L#103500;
      >=D;
      );
      A(;
      L     MD 1804;
      L     L#111600;
      <D;
      );
      O;
      A(;
      L     MD 1804;
      L     L#133500;
      >=D;
      );
      A(;
      L     MD 1804;
      L     L#141600;
      <D;
      );
      O;
      A(;
      L     MD 1804;
      L     L#163500;
      >=D;
      );
      A(;
      L     MD 1804;
      L     L#171600;
      <D;
      );
      O;
      A(;
      L     MD 1804;
      L     L#193500;
      >=D;
      );
      A(;
      L     MD 1804;
      L     L#201600;
      <D;
      );
      O;
      A(;
      L     MD 1804;
      L     L#223500;
      >=D;
      );
      A(;
      L     MD 1804;
      L     L#231600;
      <D;
      );
      O;
      A(;
      L     MD 1804;
      L     L#253500;
      >=D;
      );
      A(;
      L     MD 1804;
      L     L#261600;
      <D;
      );
      O;
      A(;
      L     MD 1804;
      L     L#283500;
      >=D;
      );
      A(;
      L     MD 1804;
      L     L#291600;
      <D;
      );
      O;
      A(;
      L     MD 1804;
      L     L#313500;
      >=D;
      );
      A(;
      L     MD 1804;
      L     L#321600;
      <D;
      );
      );
      S     #modeEmergency;
NETWORK
TITLE = STOP on carrier
      A     "ON";
      =     L 22.0;
      A     L 22.0;
      A(;
      O(;
      L     "DB_TRO"._di.MotorActPos;
      L     L#2007;
      ==D;
      );
      O(;
      L     "DB_TRO"._di.MotorActPos;
      L     L#172004;
      ==D;
      );
      );
      FP    "TRO_pFL_StopOnCarrier";
      S     "TRO_StopOnCarrier";
      A     L 22.0;
      AN    "INOUT".I_TRO.Plus;
      AN    "INOUT".I_TRO.Minus;
      R     "TRO_StopOnCarrier";
NETWORK
TITLE = Bypass mode - emergency mode for trolley
      A     "ModeBypass";
      A     "F_GBL_RECV".Signal31;
      A(;
      O     "INOUT".I_TRO.Plus;
      O     "INOUT".I_TRO.Minus;
      );
      S     #modeEmergency;
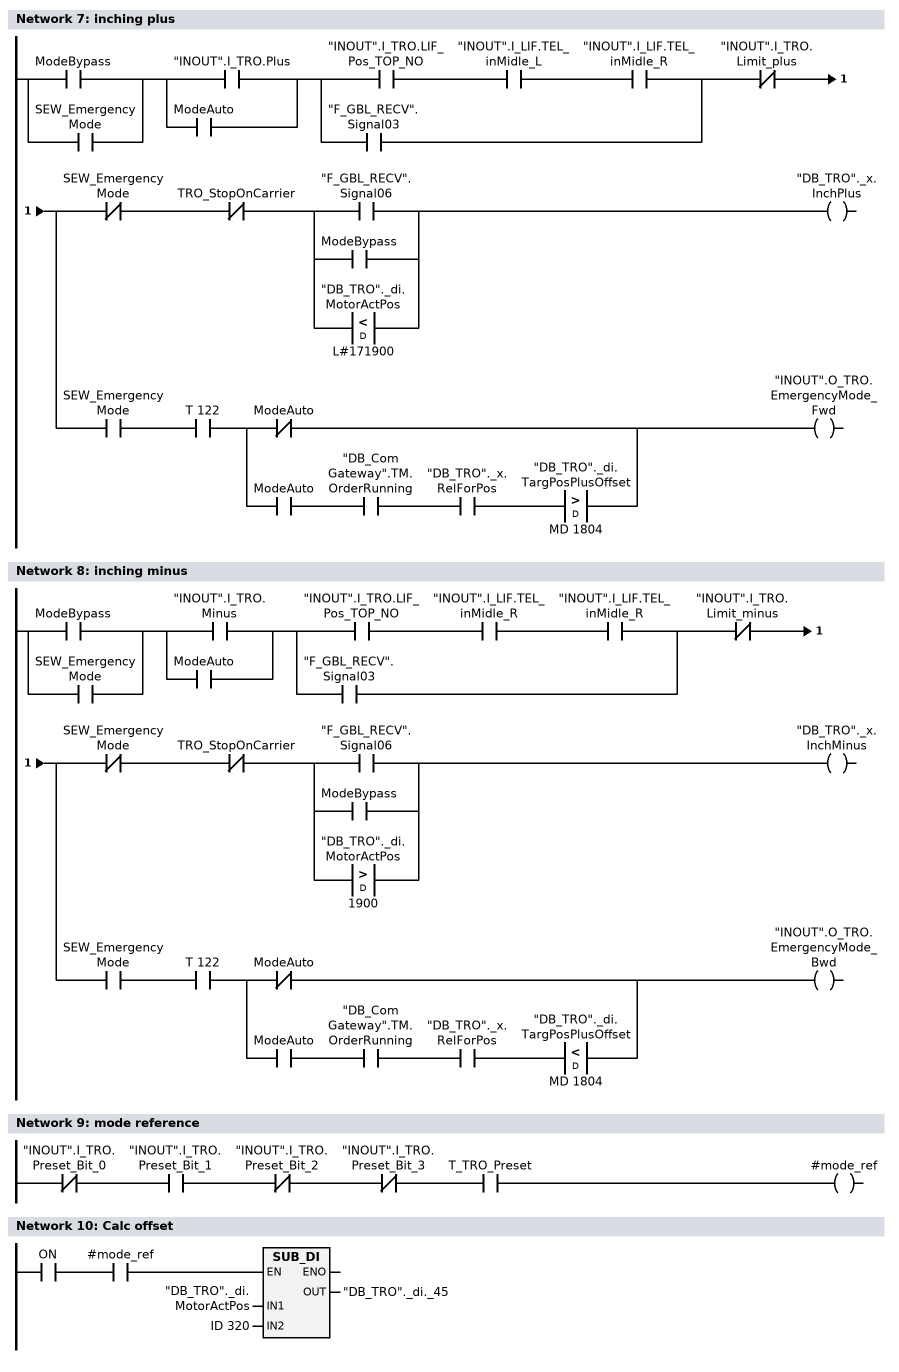
NETWORK
TITLE = inching plus
//only if service mode is not working we an use the bypass mode = JOG
      A(;
      O     "ModeBypass";
      O     "SEW_EmergencyMode";
      );
      A(;
      O     "INOUT".I_TRO.Plus;
      O     "ModeAuto";
      );
      A(;
      A     "INOUT".I_TRO.LIF_Pos_TOP_NO;
      A     "INOUT".I_LIF.TEL_inMidle_L;
      A     "INOUT".I_LIF.TEL_inMidle_R;
      O     "F_GBL_RECV".Signal03;
      );
      AN    "INOUT".I_TRO.Limit_plus;
      =     L 22.0;
      A     L 22.0;
      AN    "SEW_EmergencyMode";
      AN    "TRO_StopOnCarrier";
      A(;
      O     "F_GBL_RECV".Signal06;
      O     "ModeBypass";
      O(;
      L     "DB_TRO"._di.MotorActPos;
      L     L#171900;
      <D;
      );
      );
      =     "DB_TRO"._x.InchPlus;
      A     L 22.0;
      A     "SEW_EmergencyMode";
      A     T 122;
      A(;
      ON    "ModeAuto";
      O;
      A     "ModeAuto";
      A     "DB_ComGateway".TM.OrderRunning;
      A     "DB_TRO"._x.RelForPos;
      A(;
      L     "DB_TRO"._di.TargPosPlusOffset;
      L     MD 1804;
      >D;
      );
      );
      =     "INOUT".O_TRO.EmergencyMode_Fwd;
NETWORK
TITLE = inching minus
//only if service mode is not working we an use the bypass mode = JOG
      A(;
      O     "ModeBypass";
      O     "SEW_EmergencyMode";
      );
      A(;
      O     "INOUT".I_TRO.Minus;
      O     "ModeAuto";
      );
      A(;
      A     "INOUT".I_TRO.LIF_Pos_TOP_NO;
      A     "INOUT".I_LIF.TEL_inMidle_R;
      A     "INOUT".I_LIF.TEL_inMidle_R;
      O     "F_GBL_RECV".Signal03;
      );
      AN    "INOUT".I_TRO.Limit_minus;
      =     L 22.0;
      A     L 22.0;
      AN    "SEW_EmergencyMode";
      AN    "TRO_StopOnCarrier";
      A(;
      O     "F_GBL_RECV".Signal06;
      O     "ModeBypass";
      O(;
      L     "DB_TRO"._di.MotorActPos;
      L     1900;
      >D;
      );
      );
      =     "DB_TRO"._x.InchMinus;
      A     L 22.0;
      A     "SEW_EmergencyMode";
      A     T 122;
      A(;
      ON    "ModeAuto";
      O;
      A     "ModeAuto";
      A     "DB_ComGateway".TM.OrderRunning;
      A     "DB_TRO"._x.RelForPos;
      A(;
      L     "DB_TRO"._di.TargPosPlusOffset;
      L     MD 1804;
      <D;
      );
      );
      =     "INOUT".O_TRO.EmergencyMode_Bwd;
NETWORK
TITLE = mode reference
      AN    "INOUT".I_TRO.Preset_Bit_0;
      A     "INOUT".I_TRO.Preset_Bit_1;
      AN    "INOUT".I_TRO.Preset_Bit_2;
      AN    "INOUT".I_TRO.Preset_Bit_3;
      A     "T_TRO_Preset";
      =     #mode_ref;
NETWORK
TITLE = Calc offset
      A     "ON";
      A     #mode_ref;
      JNB   _001;
      L     "DB_TRO"._di.MotorActPos;
      L     ID 320;
      -D;
      T     "DB_TRO"._di._45;
_001: NOP   0;
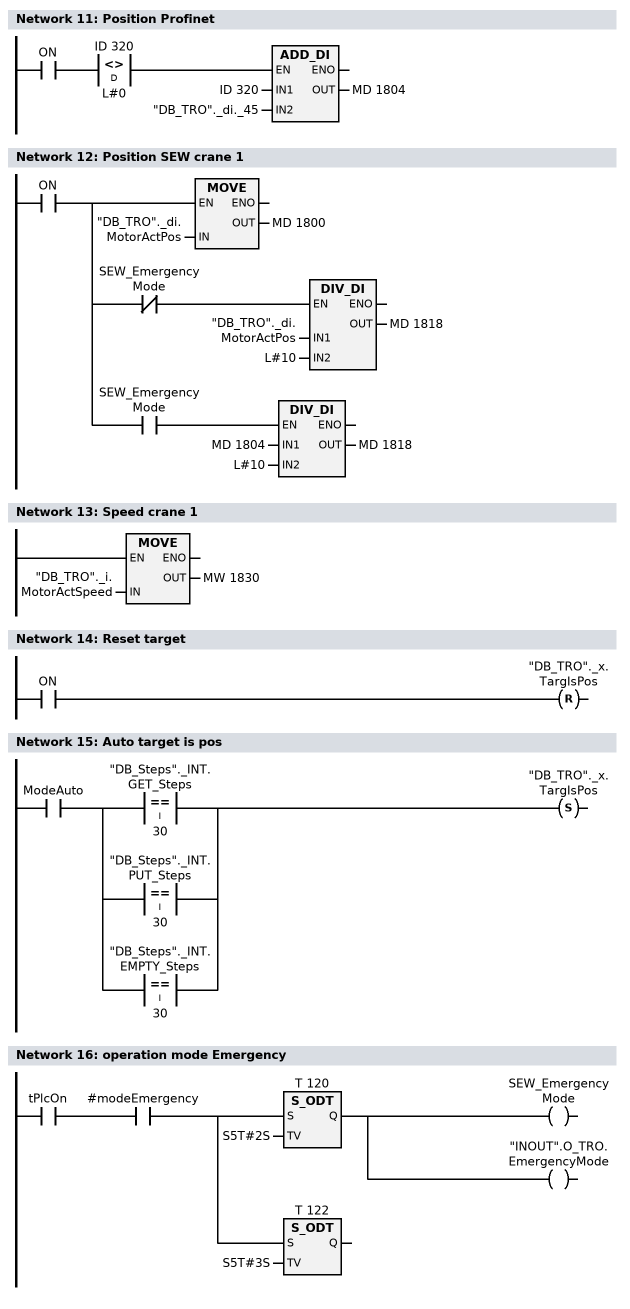
NETWORK
TITLE = Position Profinet
      A     "ON";
      A(;
      L     ID 320;
      L     L#0;
      <>D;
      );
      JNB   _002;
      L     ID 320;
      L     "DB_TRO"._di._45;
      +D;
      T     MD 1804;
_002: NOP   0;
NETWORK
TITLE = Position SEW crane 1
      A     "ON";
      =     L 22.0;
      A     L 22.0;
      JNB   _003;
      L     "DB_TRO"._di.MotorActPos;
      T     MD 1800;
_003: NOP   0;
      A     L 22.0;
      AN    "SEW_EmergencyMode";
      JNB   _004;
      L     "DB_TRO"._di.MotorActPos;
      L     L#10;
      /D;
      T     MD 1818;
_004: NOP   0;
      A     L 22.0;
      A     "SEW_EmergencyMode";
      JNB   _005;
      L     MD 1804;
      L     L#10;
      /D;
      T     MD 1818;
_005: NOP   0;
NETWORK
TITLE = Speed crane 1
      L     "DB_TRO"._i.MotorActSpeed;
      T     MW 1830;
      NOP   0;
NETWORK
TITLE = Reset target
      A     "ON";
      R     "DB_TRO"._x.TargIsPos;
NETWORK
TITLE = Auto target is pos
      A     "ModeAuto";
      A(;
      O(;
      L     "DB_Steps"._INT.GET_Steps;
      L     30;
      ==I;
      );
      O(;
      L     "DB_Steps"._INT.PUT_Steps;
      L     30;
      ==I;
      );
      O(;
      L     "DB_Steps"._INT.EMPTY_Steps;
      L     30;
      ==I;
      );
      );
      S     "DB_TRO"._x.TargIsPos;
NETWORK
TITLE = operation mode Emergency
      A     "tPlcOn";
      A     #modeEmergency;
      =     L 22.0;
      A     L 22.0;
      L     S5T#2S;
      SD    T 120;
      NOP   0;
      NOP   0;
      NOP   0;
      A     T 120;
      =     "SEW_EmergencyMode";
      =     "INOUT".O_TRO.EmergencyMode;
      A     L 22.0;
      L     S5T#3S;
      SD    T 122;
      NOP   0;
      NOP   0;
      NOP   0;
      NOP   0;
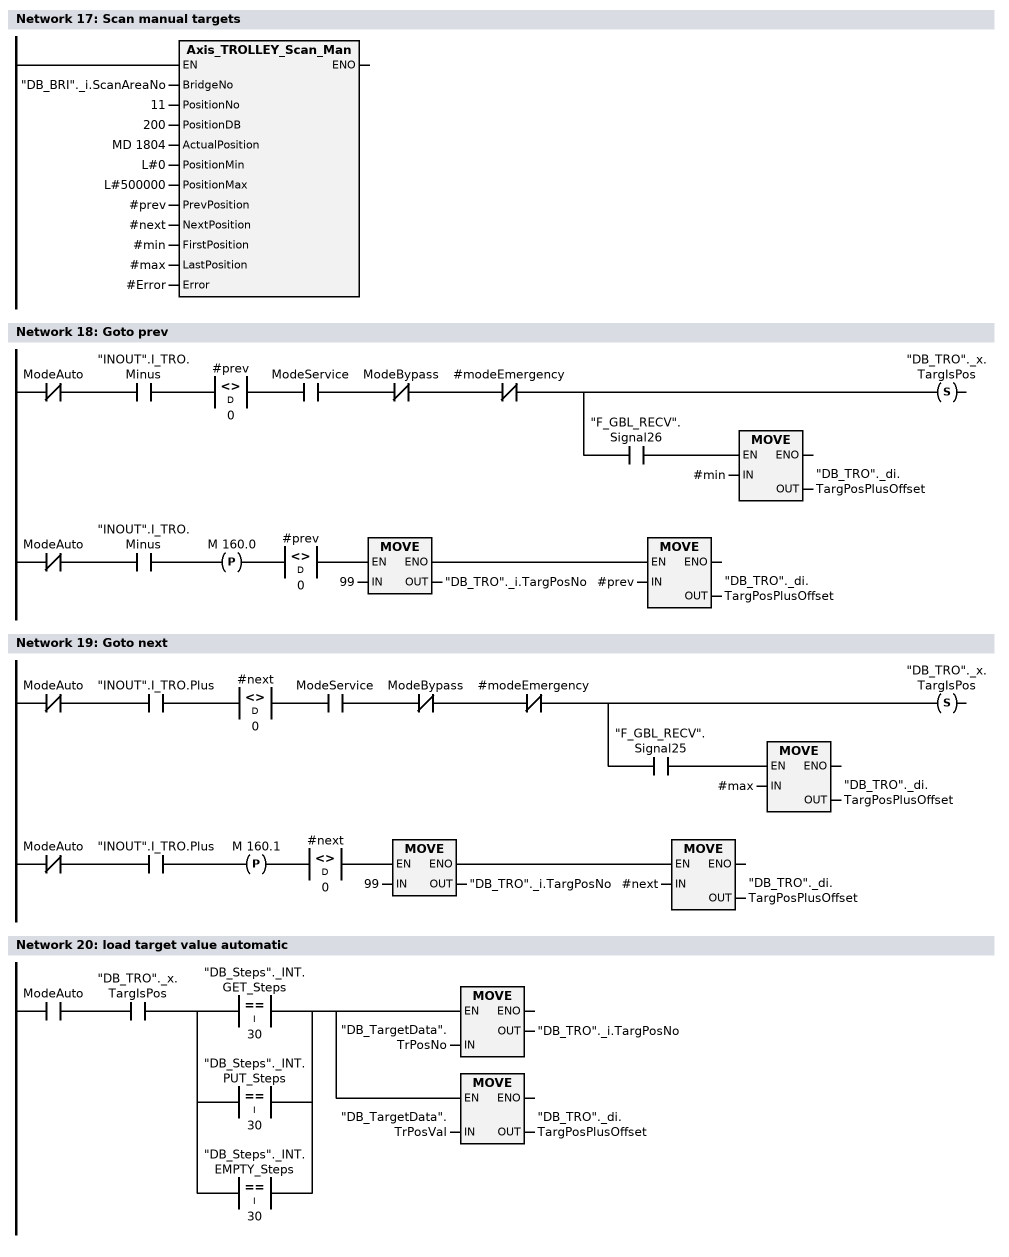
NETWORK
TITLE = Scan manual targets
      CALL  "Axis_TROLLEY_Scan_Man" (
           BridgeNo                 := "DB_BRI"._i.ScanAreaNo,
           PositionNo               := 11,
           PositionDB               := 200,
           ActualPosition           := MD 1804,
           PositionMin              := L#0,
           PositionMax              := L#500000,
           PrevPosition             := #prev,
           NextPosition             := #next,
           FirstPosition            := #min,
           LastPosition             := #max,
           Error                    := #Error);
      NOP   0;
NETWORK
TITLE = Goto prev
      AN    "ModeAuto";
      A     "INOUT".I_TRO.Minus;
      =     L 22.0;
      A(;
      A     L 22.0;
      FP    M 160.0;
      A(;
      L     #prev;
      L     0;
      <>D;
      );
      JNB   _006;
      L     99;
      T     "DB_TRO"._i.TargPosNo;
      SET;
      SAVE;
      CLR;
_006: A     BR;
      );
      JNB   _007;
      L     #prev;
      T     "DB_TRO"._di.TargPosPlusOffset;
_007: NOP   0;
      A     L 22.0;
      A(;
      L     #prev;
      L     0;
      <>D;
      );
      A     "ModeService";
      AN    "ModeBypass";
      AN    #modeEmergency;
      =     L 22.1;
      A     L 22.1;
      BLD   102;
      S     "DB_TRO"._x.TargIsPos;
      A     L 22.1;
      A     "F_GBL_RECV".Signal26;
      JNB   _008;
      L     #min;
      T     "DB_TRO"._di.TargPosPlusOffset;
_008: NOP   0;
NETWORK
TITLE = Goto next
      AN    "ModeAuto";
      A     "INOUT".I_TRO.Plus;
      =     L 22.0;
      A(;
      A     L 22.0;
      FP    M 160.1;
      A(;
      L     #next;
      L     0;
      <>D;
      );
      JNB   _009;
      L     99;
      T     "DB_TRO"._i.TargPosNo;
      SET;
      SAVE;
      CLR;
_009: A     BR;
      );
      JNB   _00a;
      L     #next;
      T     "DB_TRO"._di.TargPosPlusOffset;
_00a: NOP   0;
      A     L 22.0;
      A(;
      L     #next;
      L     0;
      <>D;
      );
      A     "ModeService";
      AN    "ModeBypass";
      AN    #modeEmergency;
      =     L 22.1;
      A     L 22.1;
      BLD   102;
      S     "DB_TRO"._x.TargIsPos;
      A     L 22.1;
      A     "F_GBL_RECV".Signal25;
      JNB   _00b;
      L     #max;
      T     "DB_TRO"._di.TargPosPlusOffset;
_00b: NOP   0;
NETWORK
TITLE = load target value automatic
      A     "ModeAuto";
      A     "DB_TRO"._x.TargIsPos;
      A(;
      O(;
      L     "DB_Steps"._INT.GET_Steps;
      L     30;
      ==I;
      );
      O(;
      L     "DB_Steps"._INT.PUT_Steps;
      L     30;
      ==I;
      );
      O(;
      L     "DB_Steps"._INT.EMPTY_Steps;
      L     30;
      ==I;
      );
      );
      =     L 22.0;
      A     L 22.0;
      JNB   _00c;
      L     "DB_TargetData".TrPosNo;
      T     "DB_TRO"._i.TargPosNo;
_00c: NOP   0;
      A     L 22.0;
      JNB   _00d;
      L     "DB_TargetData".TrPosVal;
      T     "DB_TRO"._di.TargPosPlusOffset;
_00d: NOP   0;
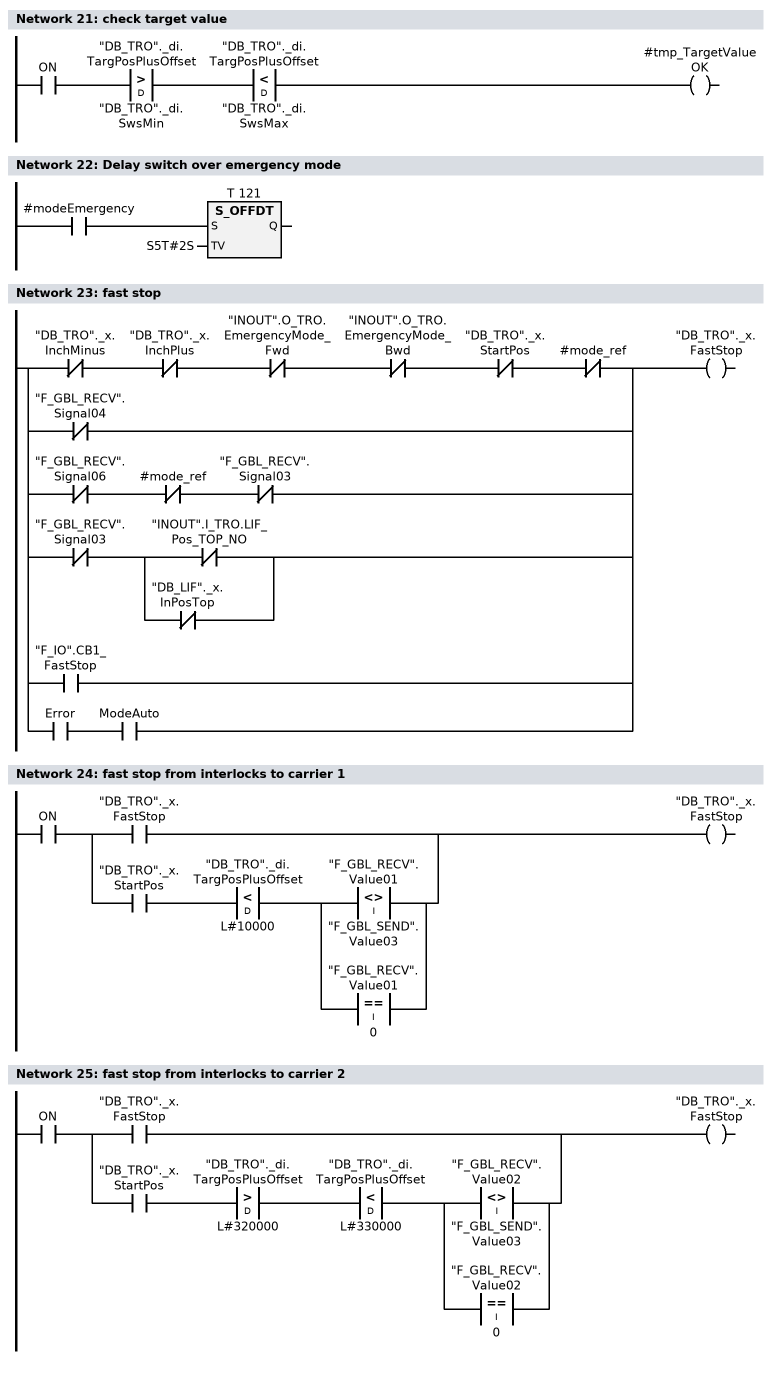
NETWORK
TITLE = check target value
      A     "ON";
      A(;
      L     "DB_TRO"._di.TargPosPlusOffset;
      L     "DB_TRO"._di.SwsMin;
      >D;
      );
      A(;
      L     "DB_TRO"._di.TargPosPlusOffset;
      L     "DB_TRO"._di.SwsMax;
      <D;
      );
      =     #tmp_TargetValueOK;
NETWORK
TITLE = Delay switch over emergency mode
      A     #modeEmergency;
      L     S5T#2S;
      SF    T 121;
      NOP   0;
      NOP   0;
      NOP   0;
      NOP   0;
NETWORK
TITLE = fast stop
      AN    "DB_TRO"._x.InchMinus;
      AN    "DB_TRO"._x.InchPlus;
      AN    "INOUT".O_TRO.EmergencyMode_Fwd;
      AN    "INOUT".O_TRO.EmergencyMode_Bwd;
      AN    "DB_TRO"._x.StartPos;
      AN    #mode_ref;
      ON    "F_GBL_RECV".Signal04;
      O;
      AN    "F_GBL_RECV".Signal06;
      AN    #mode_ref;
      AN    "F_GBL_RECV".Signal03;
      O;
      AN    "F_GBL_RECV".Signal03;
      A(;
      ON    "INOUT".I_TRO.LIF_Pos_TOP_NO;
      ON    "DB_LIF"._x.InPosTop;
      );
      O     "F_IO".CB1_FastStop;
      O;
      A     "Error";
      A     "ModeAuto";
      =     "DB_TRO"._x.FastStop;
NETWORK
TITLE = fast stop from interlocks to carrier 1
      A     "ON";
      A(;
      O     "DB_TRO"._x.FastStop;
      O;
      A     "DB_TRO"._x.StartPos;
      A(;
      L     "DB_TRO"._di.TargPosPlusOffset;
      L     L#10000;
      <D;
      );
      A(;
      O(;
      L     "F_GBL_RECV".Value01;
      L     "F_GBL_SEND".Value03;
      <>I;
      );
      O(;
      L     "F_GBL_RECV".Value01;
      L     0;
      ==I;
      );
      );
      );
      =     "DB_TRO"._x.FastStop;
NETWORK
TITLE = fast stop from interlocks to carrier 2
      A     "ON";
      A(;
      O     "DB_TRO"._x.FastStop;
      O;
      A     "DB_TRO"._x.StartPos;
      A(;
      L     "DB_TRO"._di.TargPosPlusOffset;
      L     L#320000;
      >D;
      );
      A(;
      L     "DB_TRO"._di.TargPosPlusOffset;
      L     L#330000;
      <D;
      );
      A(;
      O(;
      L     "F_GBL_RECV".Value02;
      L     "F_GBL_SEND".Value03;
      <>I;
      );
      O(;
      L     "F_GBL_RECV".Value02;
      L     0;
      ==I;
      );
      );
      );
      =     "DB_TRO"._x.FastStop;
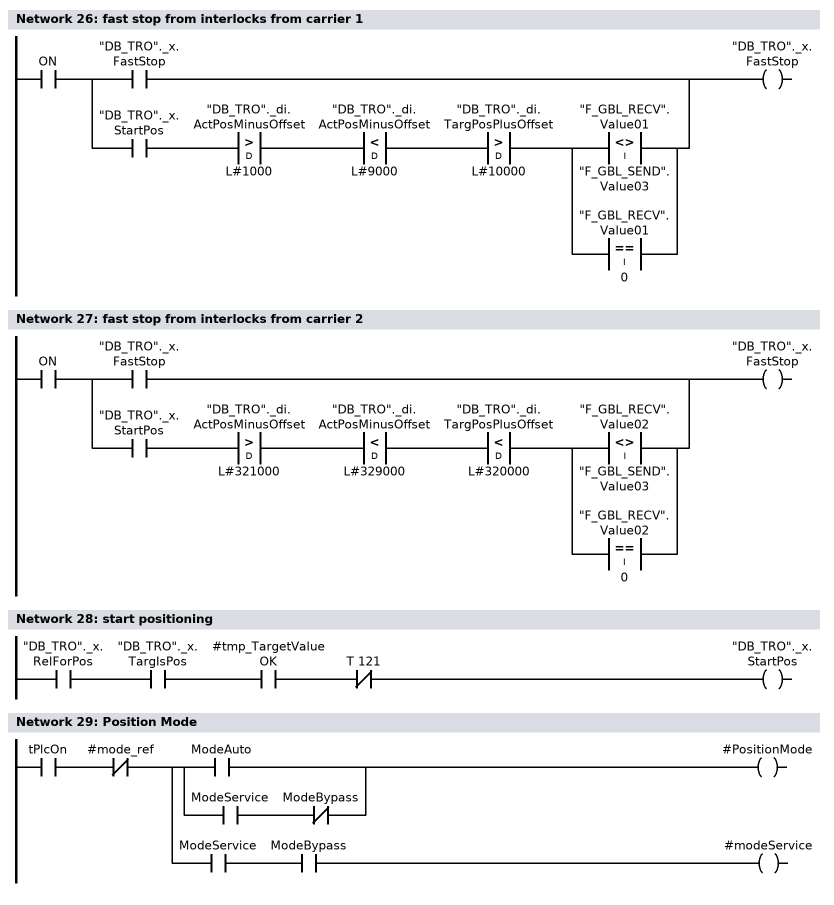
NETWORK
TITLE = fast stop from interlocks from carrier 1
      A     "ON";
      A(;
      O     "DB_TRO"._x.FastStop;
      O;
      A     "DB_TRO"._x.StartPos;
      A(;
      L     "DB_TRO"._di.ActPosMinusOffset;
      L     L#1000;
      >D;
      );
      A(;
      L     "DB_TRO"._di.ActPosMinusOffset;
      L     L#9000;
      <D;
      );
      A(;
      L     "DB_TRO"._di.TargPosPlusOffset;
      L     L#10000;
      >D;
      );
      A(;
      O(;
      L     "F_GBL_RECV".Value01;
      L     "F_GBL_SEND".Value03;
      <>I;
      );
      O(;
      L     "F_GBL_RECV".Value01;
      L     0;
      ==I;
      );
      );
      );
      =     "DB_TRO"._x.FastStop;
NETWORK
TITLE = fast stop from interlocks from carrier 2
      A     "ON";
      A(;
      O     "DB_TRO"._x.FastStop;
      O;
      A     "DB_TRO"._x.StartPos;
      A(;
      L     "DB_TRO"._di.ActPosMinusOffset;
      L     L#321000;
      >D;
      );
      A(;
      L     "DB_TRO"._di.ActPosMinusOffset;
      L     L#329000;
      <D;
      );
      A(;
      L     "DB_TRO"._di.TargPosPlusOffset;
      L     L#320000;
      <D;
      );
      A(;
      O(;
      L     "F_GBL_RECV".Value02;
      L     "F_GBL_SEND".Value03;
      <>I;
      );
      O(;
      L     "F_GBL_RECV".Value02;
      L     0;
      ==I;
      );
      );
      );
      =     "DB_TRO"._x.FastStop;
NETWORK
TITLE = start positioning
      A     "DB_TRO"._x.RelForPos;
      A     "DB_TRO"._x.TargIsPos;
      A     #tmp_TargetValueOK;
      AN    T 121;
      =     "DB_TRO"._x.StartPos;
NETWORK
TITLE = Position Mode
      A     "tPlcOn";
      AN    #mode_ref;
      =     L 22.0;
      A     L 22.0;
      A(;
      O     "ModeAuto";
      O;
      A     "ModeService";
      AN    "ModeBypass";
      );
      =     #PositionMode;
      A     L 22.0;
      A     "ModeService";
      A     "ModeBypass";
      =     #modeService;
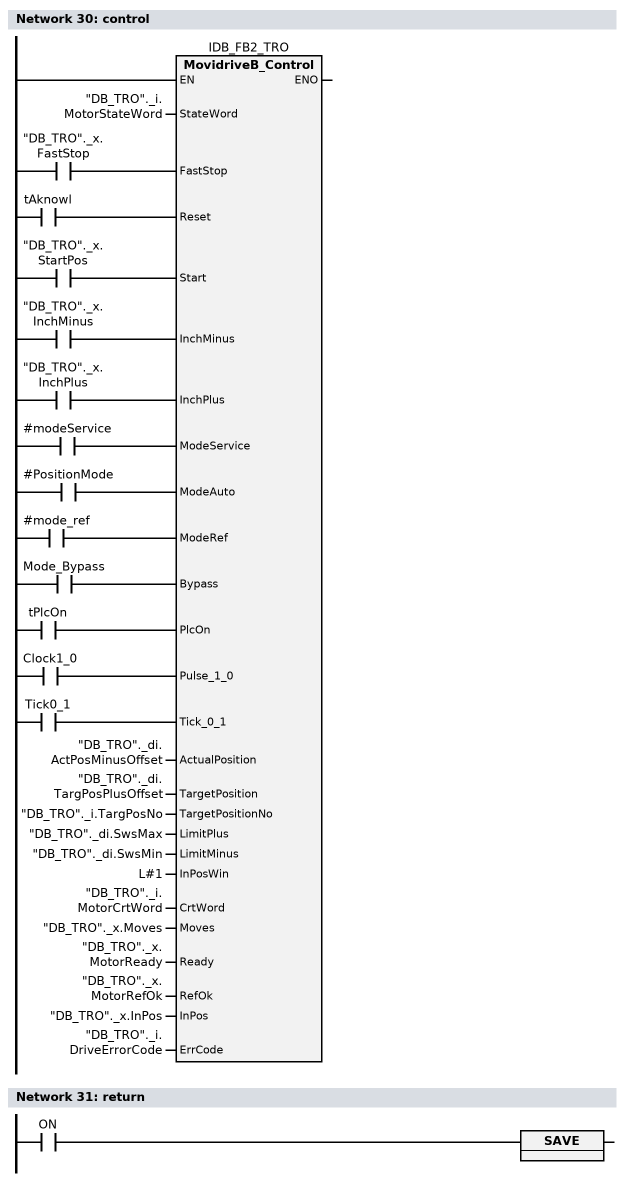
NETWORK
TITLE = control
      A     "DB_TRO"._x.FastStop;
      =     L 22.0;
      BLD   103;
      A     "tAknowl";
      =     L 22.1;
      BLD   103;
      A     "DB_TRO"._x.StartPos;
      =     L 22.2;
      BLD   103;
      A     "DB_TRO"._x.InchMinus;
      =     L 22.3;
      BLD   103;
      A     "DB_TRO"._x.InchPlus;
      =     L 22.4;
      BLD   103;
      A     #modeService;
      =     L 22.5;
      BLD   103;
      A     #PositionMode;
      =     L 22.6;
      BLD   103;
      A     #mode_ref;
      =     L 22.7;
      BLD   103;
      A     "Mode_Bypass";
      =     L 23.0;
      BLD   103;
      A     "tPlcOn";
      =     L 23.1;
      BLD   103;
      A     "Clock1_0";
      =     L 23.2;
      BLD   103;
      A     "Tick0_1";
      =     L 23.3;
      BLD   103;
      CALL  "MovidriveB_Control" , "IDB_FB2_TRO" (
           StateWord                := "DB_TRO"._i.MotorStateWord,
           FastStop                 := L 22.0,
           Reset                    := L 22.1,
           Start                    := L 22.2,
           InchMinus                := L 22.3,
           InchPlus                 := L 22.4,
           ModeService              := L 22.5,
           ModeAuto                 := L 22.6,
           ModeRef                  := L 22.7,
           Bypass                   := L 23.0,
           PlcOn                    := L 23.1,
           Pulse_1_0                := L 23.2,
           Tick_0_1                 := L 23.3,
           ActualPosition           := "DB_TRO"._di.ActPosMinusOffset,
           TargetPosition           := "DB_TRO"._di.TargPosPlusOffset,
           TargetPositionNo         := "DB_TRO"._i.TargPosNo,
           LimitPlus                := "DB_TRO"._di.SwsMax,
           LimitMinus               := "DB_TRO"._di.SwsMin,
           InPosWin                 := L#1,
           CrtWord                  := "DB_TRO"._i.MotorCrtWord,
           Moves                    := "DB_TRO"._x.Moves,
           Ready                    := "DB_TRO"._x.MotorReady,
           RefOk                    := "DB_TRO"._x.MotorRefOk,
           InPos                    := "DB_TRO"._x.InPos,
           ErrCode                  := "DB_TRO"._i.DriveErrorCode);
      NOP   0;
NETWORK
TITLE = return
      A     "ON";
      SAVE;
END_FUNCTION

FUNCTION "Axis_TROLLEY_Speed" : VOID	// FC 213
TITLE = TROLLEY Speed
VERSION : 0.1
VAR_TEMP
  tmp_di_1 : DINT ;
  tmp_di_2 : DINT ;
  tmp_i_1 : INT ;
  tmp_i_2 : INT ;
  tmp_speed : INT ;
END_VAR
BEGIN
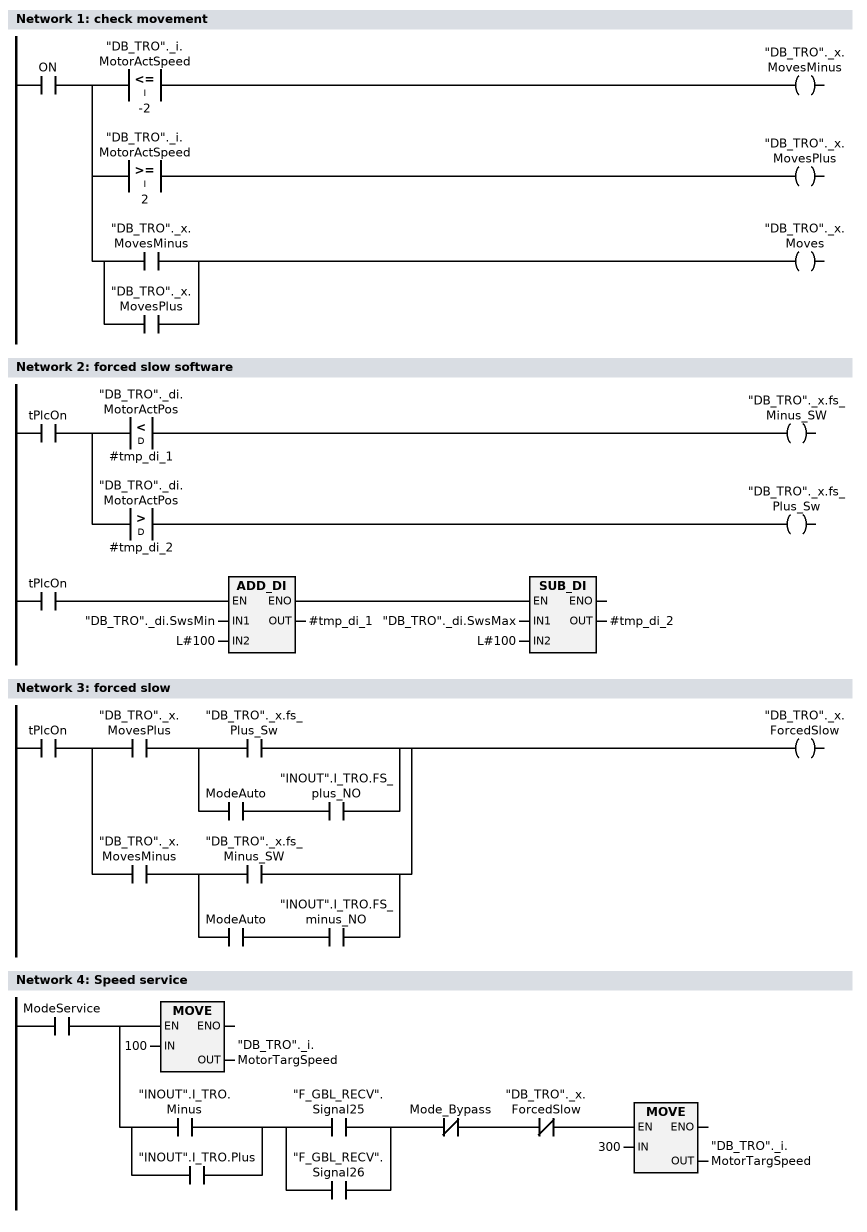
NETWORK
TITLE = check movement
      A     "ON";
      =     L 14.0;
      A     L 14.0;
      A(;
      L     "DB_TRO"._i.MotorActSpeed;
      L     -2;
      <=I;
      );
      =     "DB_TRO"._x.MovesMinus;
      A     L 14.0;
      A(;
      L     "DB_TRO"._i.MotorActSpeed;
      L     2;
      >=I;
      );
      =     "DB_TRO"._x.MovesPlus;
      A     L 14.0;
      A(;
      O     "DB_TRO"._x.MovesMinus;
      O     "DB_TRO"._x.MovesPlus;
      );
      =     "DB_TRO"._x.Moves;
NETWORK
TITLE = forced slow software
      A     "tPlcOn";
      =     L 14.0;
      A(;
      A     L 14.0;
      JNB   _001;
      L     "DB_TRO"._di.SwsMin;
      L     L#100;
      +D;
      T     #tmp_di_1;
      AN    OV;
      SAVE;
      CLR;
_001: A     BR;
      );
      JNB   _002;
      L     "DB_TRO"._di.SwsMax;
      L     L#100;
      -D;
      T     #tmp_di_2;
_002: NOP   0;
      A     L 14.0;
      A(;
      L     "DB_TRO"._di.MotorActPos;
      L     #tmp_di_1;
      <D;
      );
      =     "DB_TRO"._x.fs_Minus_SW;
      A     L 14.0;
      A(;
      L     "DB_TRO"._di.MotorActPos;
      L     #tmp_di_2;
      >D;
      );
      =     "DB_TRO"._x.fs_Plus_Sw;
NETWORK
TITLE = forced slow
//in service we use only the software, in auto we use the prox. switches
      A     "tPlcOn";
      A(;
      A     "DB_TRO"._x.MovesPlus;
      A(;
      O     "DB_TRO"._x.fs_Plus_Sw;
      O;
      A     "ModeAuto";
      A     "INOUT".I_TRO.FS_plus_NO;
      );
      O;
      A     "DB_TRO"._x.MovesMinus;
      A(;
      O     "DB_TRO"._x.fs_Minus_SW;
      O;
      A     "ModeAuto";
      A     "INOUT".I_TRO.FS_minus_NO;
      );
      );
      =     "DB_TRO"._x.ForcedSlow;
NETWORK
TITLE = Speed service
//in bypass we do not allow faster speed
//Fast old: 150
      A     "ModeService";
      =     L 14.0;
      A     L 14.0;
      JNB   _003;
      L     100;
      T     "DB_TRO"._i.MotorTargSpeed;
_003: NOP   0;
      A     L 14.0;
      A(;
      O     "INOUT".I_TRO.Minus;
      O     "INOUT".I_TRO.Plus;
      );
      A(;
      O     "F_GBL_RECV".Signal25;
      O     "F_GBL_RECV".Signal26;
      );
      AN    "Mode_Bypass";
      AN    "DB_TRO"._x.ForcedSlow;
      JNB   _004;
      L     300;
      T     "DB_TRO"._i.MotorTargSpeed;
_004: NOP   0;
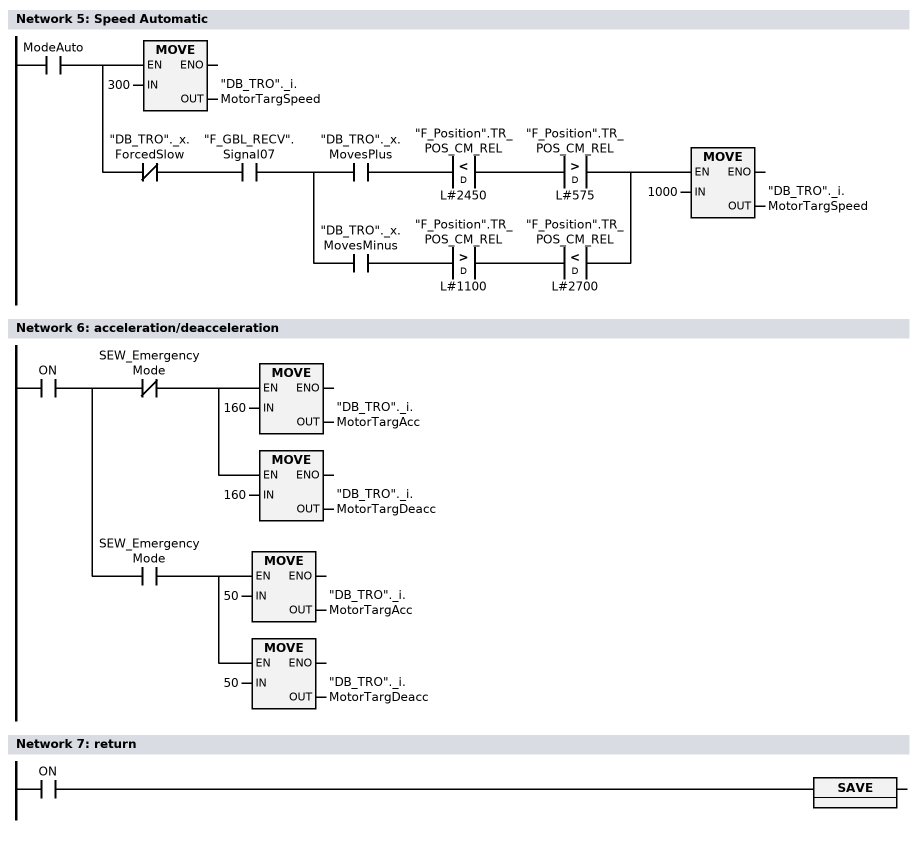
NETWORK
TITLE = Speed Automatic
//speed was 1200
//
      A     "ModeAuto";
      =     L 14.0;
      A     L 14.0;
      JNB   _005;
      L     300;
      T     "DB_TRO"._i.MotorTargSpeed;
_005: NOP   0;
      A     L 14.0;
      AN    "DB_TRO"._x.ForcedSlow;
      A     "F_GBL_RECV".Signal07;
      A(;
      A     "DB_TRO"._x.MovesPlus;
      A(;
      L     "F_Position".TR_POS_CM_REL;
      L     L#2450;
      <D;
      );
      A(;
      L     "F_Position".TR_POS_CM_REL;
      L     L#575;
      >D;
      );
      O;
      A     "DB_TRO"._x.MovesMinus;
      A(;
      L     "F_Position".TR_POS_CM_REL;
      L     L#1100;
      >D;
      );
      A(;
      L     "F_Position".TR_POS_CM_REL;
      L     L#2700;
      <D;
      );
      );
      JNB   _006;
      L     1000;
      T     "DB_TRO"._i.MotorTargSpeed;
_006: NOP   0;
NETWORK
TITLE = acceleration/deacceleration
//acc/dec was 2000
      A     "ON";
      =     L 14.0;
      A     L 14.0;
      AN    "SEW_EmergencyMode";
      =     L 14.1;
      A     L 14.1;
      JNB   _007;
      L     160;
      T     "DB_TRO"._i.MotorTargAcc;
_007: NOP   0;
      A     L 14.1;
      JNB   _008;
      L     160;
      T     "DB_TRO"._i.MotorTargDeacc;
_008: NOP   0;
      A     L 14.0;
      A     "SEW_EmergencyMode";
      =     L 14.1;
      A     L 14.1;
      JNB   _009;
      L     50;
      T     "DB_TRO"._i.MotorTargAcc;
_009: NOP   0;
      A     L 14.1;
      JNB   _00a;
      L     50;
      T     "DB_TRO"._i.MotorTargDeacc;
_00a: NOP   0;
NETWORK
TITLE = return
      A     "ON";
      SAVE;
END_FUNCTION

FUNCTION "Axis_TROLLEY_Scan" : VOID	// FC 214
TITLE = TROLLEY Scan
VERSION : 0.1
VAR_TEMP
  tmp_di_1 : DINT ;
  tmp_di_PosWin : DINT ;
  tmp_i_BRIScanSetNo : INT ;
  tmp_i_LIF_DBNo : INT ;
  tmp_i_LIF_DBNo_2 : INT ;
  tmp_di_Scan_Pos : DINT ;
  tmp_di_Scan_Plus : DINT ;
  tmp_di_Scan_Minus : DINT ;
  startValue : DINT ;
  brNo : INT ;
  NoDB : INT ;
  retVal : INT ;
  start : BOOL ;
  pMem : DINT ;
  trNo : INT ;
END_VAR
BEGIN
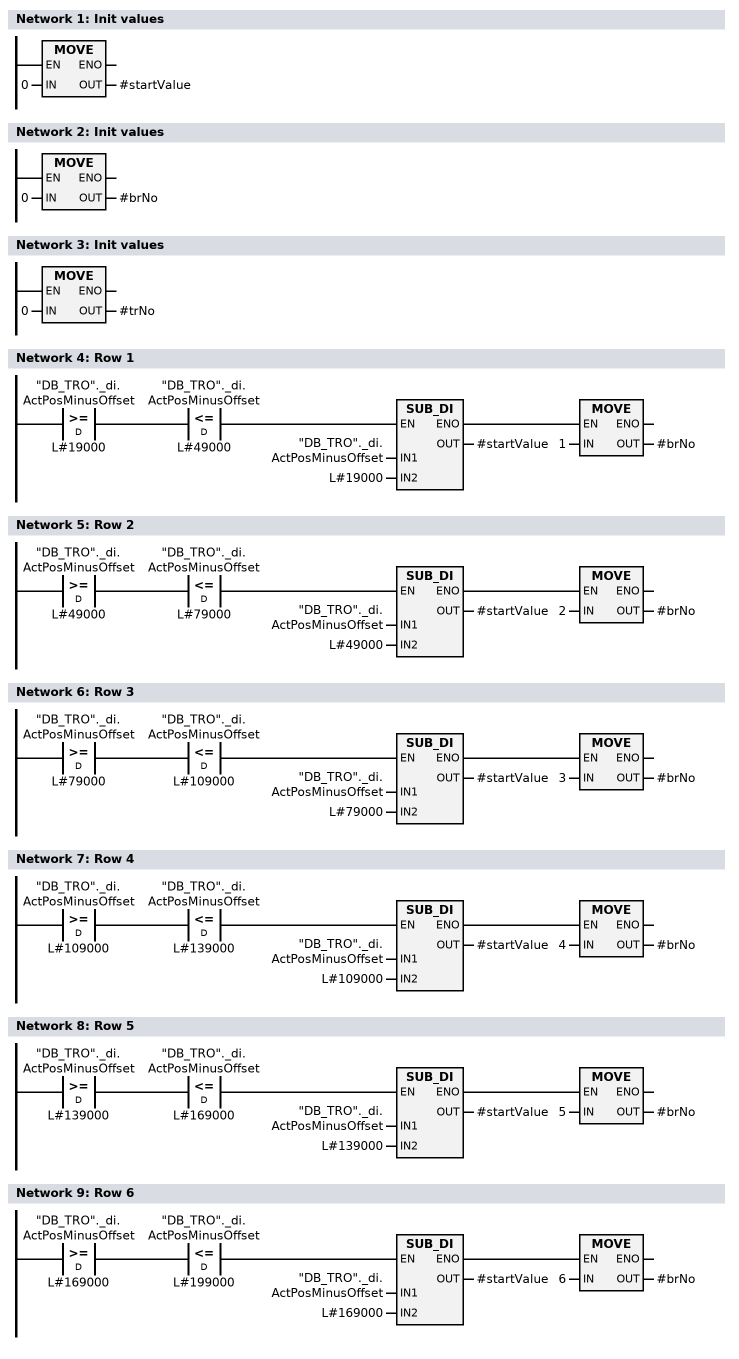
NETWORK
TITLE = Init values
      L     0;
      T     #startValue;
      NOP   0;
NETWORK
TITLE = Init values
      L     0;
      T     #brNo;
      NOP   0;
NETWORK
TITLE = Init values
      L     0;
      T     #trNo;
      NOP   0;
NETWORK
TITLE = Row 1
      A(;
      A(;
      L     "DB_TRO"._di.ActPosMinusOffset;
      L     L#19000;
      >=D;
      );
      A(;
      L     "DB_TRO"._di.ActPosMinusOffset;
      L     L#49000;
      <=D;
      );
      JNB   _001;
      L     "DB_TRO"._di.ActPosMinusOffset;
      L     L#19000;
      -D;
      T     #startValue;
      AN    OV;
      SAVE;
      CLR;
_001: A     BR;
      );
      JNB   _002;
      L     1;
      T     #brNo;
_002: NOP   0;
NETWORK
TITLE = Row 2
      A(;
      A(;
      L     "DB_TRO"._di.ActPosMinusOffset;
      L     L#49000;
      >=D;
      );
      A(;
      L     "DB_TRO"._di.ActPosMinusOffset;
      L     L#79000;
      <=D;
      );
      JNB   _003;
      L     "DB_TRO"._di.ActPosMinusOffset;
      L     L#49000;
      -D;
      T     #startValue;
      AN    OV;
      SAVE;
      CLR;
_003: A     BR;
      );
      JNB   _004;
      L     2;
      T     #brNo;
_004: NOP   0;
NETWORK
TITLE = Row 3
      A(;
      A(;
      L     "DB_TRO"._di.ActPosMinusOffset;
      L     L#79000;
      >=D;
      );
      A(;
      L     "DB_TRO"._di.ActPosMinusOffset;
      L     L#109000;
      <=D;
      );
      JNB   _005;
      L     "DB_TRO"._di.ActPosMinusOffset;
      L     L#79000;
      -D;
      T     #startValue;
      AN    OV;
      SAVE;
      CLR;
_005: A     BR;
      );
      JNB   _006;
      L     3;
      T     #brNo;
_006: NOP   0;
NETWORK
TITLE = Row 4
      A(;
      A(;
      L     "DB_TRO"._di.ActPosMinusOffset;
      L     L#109000;
      >=D;
      );
      A(;
      L     "DB_TRO"._di.ActPosMinusOffset;
      L     L#139000;
      <=D;
      );
      JNB   _007;
      L     "DB_TRO"._di.ActPosMinusOffset;
      L     L#109000;
      -D;
      T     #startValue;
      AN    OV;
      SAVE;
      CLR;
_007: A     BR;
      );
      JNB   _008;
      L     4;
      T     #brNo;
_008: NOP   0;
NETWORK
TITLE = Row 5
      A(;
      A(;
      L     "DB_TRO"._di.ActPosMinusOffset;
      L     L#139000;
      >=D;
      );
      A(;
      L     "DB_TRO"._di.ActPosMinusOffset;
      L     L#169000;
      <=D;
      );
      JNB   _009;
      L     "DB_TRO"._di.ActPosMinusOffset;
      L     L#139000;
      -D;
      T     #startValue;
      AN    OV;
      SAVE;
      CLR;
_009: A     BR;
      );
      JNB   _00a;
      L     5;
      T     #brNo;
_00a: NOP   0;
NETWORK
TITLE = Row 6
      A(;
      A(;
      L     "DB_TRO"._di.ActPosMinusOffset;
      L     L#169000;
      >=D;
      );
      A(;
      L     "DB_TRO"._di.ActPosMinusOffset;
      L     L#199000;
      <=D;
      );
      JNB   _00b;
      L     "DB_TRO"._di.ActPosMinusOffset;
      L     L#169000;
      -D;
      T     #startValue;
      AN    OV;
      SAVE;
      CLR;
_00b: A     BR;
      );
      JNB   _00c;
      L     6;
      T     #brNo;
_00c: NOP   0;
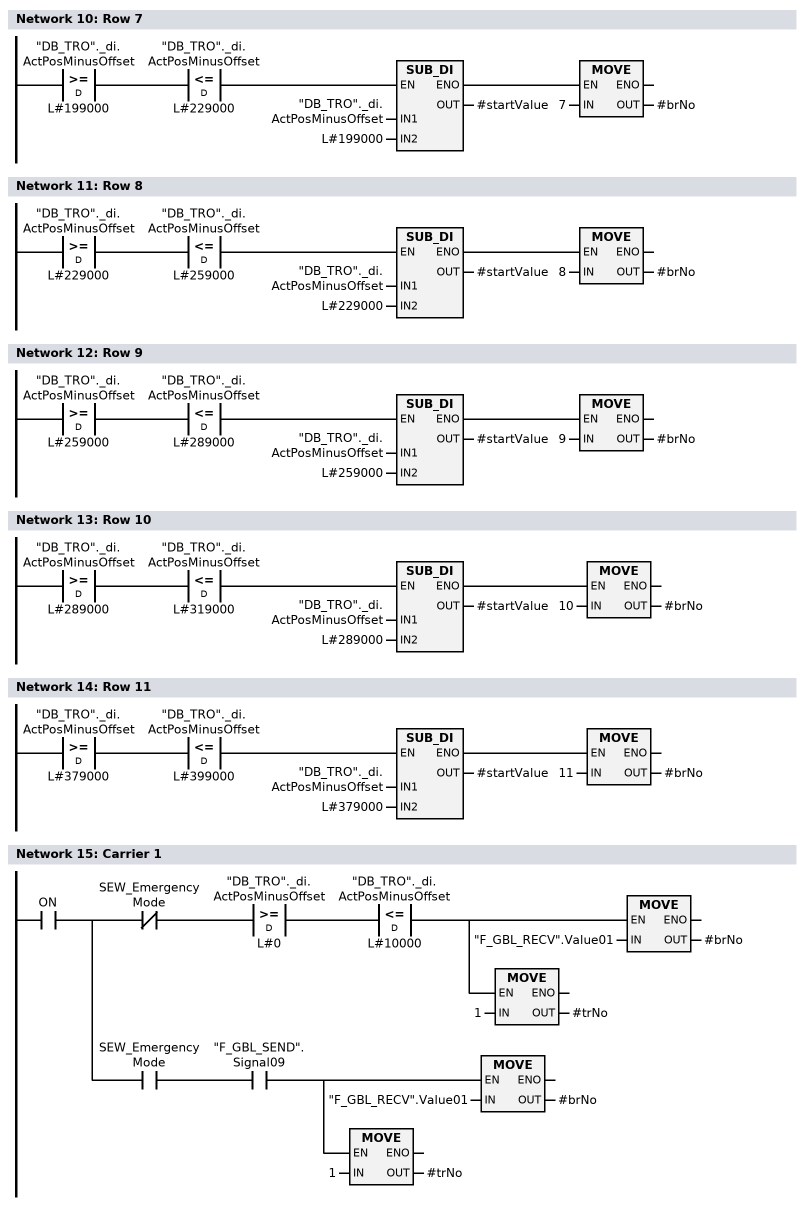
NETWORK
TITLE = Row 7
      A(;
      A(;
      L     "DB_TRO"._di.ActPosMinusOffset;
      L     L#199000;
      >=D;
      );
      A(;
      L     "DB_TRO"._di.ActPosMinusOffset;
      L     L#229000;
      <=D;
      );
      JNB   _00d;
      L     "DB_TRO"._di.ActPosMinusOffset;
      L     L#199000;
      -D;
      T     #startValue;
      AN    OV;
      SAVE;
      CLR;
_00d: A     BR;
      );
      JNB   _00e;
      L     7;
      T     #brNo;
_00e: NOP   0;
NETWORK
TITLE = Row 8
      A(;
      A(;
      L     "DB_TRO"._di.ActPosMinusOffset;
      L     L#229000;
      >=D;
      );
      A(;
      L     "DB_TRO"._di.ActPosMinusOffset;
      L     L#259000;
      <=D;
      );
      JNB   _00f;
      L     "DB_TRO"._di.ActPosMinusOffset;
      L     L#229000;
      -D;
      T     #startValue;
      AN    OV;
      SAVE;
      CLR;
_00f: A     BR;
      );
      JNB   _010;
      L     8;
      T     #brNo;
_010: NOP   0;
NETWORK
TITLE = Row 9
      A(;
      A(;
      L     "DB_TRO"._di.ActPosMinusOffset;
      L     L#259000;
      >=D;
      );
      A(;
      L     "DB_TRO"._di.ActPosMinusOffset;
      L     L#289000;
      <=D;
      );
      JNB   _011;
      L     "DB_TRO"._di.ActPosMinusOffset;
      L     L#259000;
      -D;
      T     #startValue;
      AN    OV;
      SAVE;
      CLR;
_011: A     BR;
      );
      JNB   _012;
      L     9;
      T     #brNo;
_012: NOP   0;
NETWORK
TITLE = Row 10
      A(;
      A(;
      L     "DB_TRO"._di.ActPosMinusOffset;
      L     L#289000;
      >=D;
      );
      A(;
      L     "DB_TRO"._di.ActPosMinusOffset;
      L     L#319000;
      <=D;
      );
      JNB   _013;
      L     "DB_TRO"._di.ActPosMinusOffset;
      L     L#289000;
      -D;
      T     #startValue;
      AN    OV;
      SAVE;
      CLR;
_013: A     BR;
      );
      JNB   _014;
      L     10;
      T     #brNo;
_014: NOP   0;
NETWORK
TITLE = Row 11
      A(;
      A(;
      L     "DB_TRO"._di.ActPosMinusOffset;
      L     L#379000;
      >=D;
      );
      A(;
      L     "DB_TRO"._di.ActPosMinusOffset;
      L     L#399000;
      <=D;
      );
      JNB   _015;
      L     "DB_TRO"._di.ActPosMinusOffset;
      L     L#379000;
      -D;
      T     #startValue;
      AN    OV;
      SAVE;
      CLR;
_015: A     BR;
      );
      JNB   _016;
      L     11;
      T     #brNo;
_016: NOP   0;
NETWORK
TITLE = Carrier 1
      A     "ON";
      =     L 44.0;
      A     L 44.0;
      AN    "SEW_EmergencyMode";
      A(;
      L     "DB_TRO"._di.ActPosMinusOffset;
      L     L#0;
      >=D;
      );
      A(;
      L     "DB_TRO"._di.ActPosMinusOffset;
      L     L#10000;
      <=D;
      );
      =     L 44.1;
      A     L 44.1;
      JNB   _017;
      L     "F_GBL_RECV".Value01;
      T     #brNo;
_017: NOP   0;
      A     L 44.1;
      JNB   _018;
      L     1;
      T     #trNo;
_018: NOP   0;
      A     L 44.0;
      A     "SEW_EmergencyMode";
      A     "F_GBL_SEND".Signal09;
      =     L 44.1;
      A     L 44.1;
      JNB   _019;
      L     "F_GBL_RECV".Value01;
      T     #brNo;
_019: NOP   0;
      A     L 44.1;
      JNB   _01a;
      L     1;
      T     #trNo;
_01a: NOP   0;
